// ---- ECC/Basic/TrackClient/Node Data/ST_ReadStationData.TcDUT
{attribute 'pack_mode' := '1'}
TYPE ST_ReadStationData :
STRUCT
	stReadListReturnInfo		: ARRAY [1..1] OF ST_UAReadListReturnInfo;
	stStationData				: ST_StatusStation;

END_STRUCT
END_TYPE

// ---- ECC/Basic/TrackClient/Node Data/ST_ReadVehicleData.TcDUT
{attribute 'pack_mode' := '1'}
TYPE ST_ReadVehicleData :
STRUCT
	stReadListReturnInfo		: ARRAY [1..1] OF ST_UAReadListReturnInfo;
	stVehicle					: ST_StatusVehicle;

END_STRUCT
END_TYPE

// ---- ECC/Basic/TrackClient/Node Data/ST_ReadVehicleData_OLD.TcDUT
{attribute 'pack_mode' := '1'}
TYPE ST_ReadVehicleData_OLD :
STRUCT
//	stReadListReturnInfo		: ARRAY [1..1] OF ST_UAReadListReturnInfo;
//	stVehicle					: ST_StatusVehicle;

	// Array must have the same number as the amount of elements in the status strucuture! 
	stReadListReturnInfo		: ARRAY [1..8] OF ST_UAReadListReturnInfo;
	nVehicleID					: UINT;
	bVehiclePresent				: BOOL;
	nState						: UINT; 
	nPathID						: UINT;
	fPosition					: REAL;
	nTargetPathID				: UINT;
	fTargetPosition				: REAL;
	fVelocity					: REAL;
END_STRUCT
END_TYPE

// ---- ECC/Basic/TrackClient/Node Data/ST_StatusCell.TcDUT
/// Standard Status for cells
TYPE ST_StatusCell :
STRUCT
	sCellID						: STRING(30);		(*  *)
	sNextCellOnTrack			: STRING(30);		(*  *)
//	nVehicleIDDecisionPoint		: UINT;				(* ID of the vehicle ready at cell decision point *)
//													(* ZERO of no vehicle is ready *)	
//	sCarrierIDDecisionPoint		: STRING(30);		(* ID of the carrier ready at cell decision point *)
	astReservations				: ARRAY [1..MM_MAX_RESERVATIONLIST_ELEMENTS] OF ST_ReservationData; (* Reservation lists for cells. *)
																									(* NOTE! Only manipulated through methods M_AddReservationList, M_RemoveReservationList *)
	anVehicles					: ARRAY [1..MM_MAX_NUMBER_OF_VEHICLE_ELEMENTS] OF UINT;				(* Vehicles ID's of the vehicles controlled by this cell *)

END_STRUCT
END_TYPE

// ---- ECC/Basic/TrackClient/Node Data/ST_StatusNode.TcDUT
{attribute 'pack_mode' := '1'}
TYPE ST_StatusNode :
STRUCT
	nState	: UINT;
	rTemp	: REAL;
END_STRUCT
END_TYPE

// ---- ECC/Basic/TrackClient/Node Data/ST_StatusPath.TcDUT
{attribute 'pack_mode' := '1'}
TYPE ST_StatusPath :
STRUCT
	nPathID						: UINT;
	sCellID						: STRING(30);
	bPathPresent				: BOOL;
	nState						: UINT;			// E_MMPathState
	nMotionStatus				: UINT;			// E_MMPathMotionStatus
END_STRUCT
END_TYPE

// ---- ECC/Basic/TrackClient/Node Data/ST_StatusStation.TcDUT
{attribute 'pack_mode' := '1'}
TYPE ST_StatusStation :
STRUCT
	sCellID						: STRING(30);
	sStationID					: STRING(30);
	bStationPresent				: BOOL;
	nVehicleIDDecisionPoint		: UINT;				(* ID of the vehicle ready at station decision point. ZERO of no vehicle is ready *)	
	sCarrierIDDecisionPoint		: STRING(30);		(* ID of the carrier ready at station decision point *)
	nVehicleIDStationIn			: UINT;				(* ID of the vehicle ready at station location In location. ZERO of no vehicle is ready *)	
	sCarrierIDStationIn			: STRING(30);		(* ID of the carrier ready at station location In location *)
	nVehicleIDStationOut		: UINT;				(* ID of the vehicle ready at station location Out ZERO of no vehicle is ready *)	
	sCarrierIDStationOut		: STRING(30);		(* ID of the carrier ready at station location Out location *)
//	stStation					: ST_StatusBuffer;
//	aPreBuffer					: ARRAY [1..MM_MAX_BUFFER_INDEX] OF ST_StatusBuffer;
//	aPostBuffer					: ARRAY [1..MM_MAX_BUFFER_INDEX] OF ST_StatusBuffer;

END_STRUCT
END_TYPE

// ---- ECC/Basic/TrackClient/Node Data/ST_StatusVehicle.TcDUT
{attribute 'pack_mode' := '1'}
TYPE ST_StatusVehicle :
STRUCT
	nVehicleID					: UINT;
	sOwnerCell					: STRING(30);				// Cell which controls this vehicle
	nState						: UINT;						// E_CarrierStatus: 0: Undefined, 1: Initiating, 2: Not Busy(No Ticket), 3: Busy(Ticket), 4: Montage Reserved
	bVehiclePresent				: BOOL;
	bDataValid					: BOOL;
	sLastScan					: STRING(30);				// Timestamp for last scan of this vehicle
	sCarrierID					: STRING(30);				// Scanned (from Carrier RFID scan)
	bTool						: BOOL;						// TRUE if tool is mounted on carrier
	sToolID						: STRING(30);				// Tool ID (if mounted) (from Tool RFID scan)
	bMaterial					: BOOL;						// TRUE if material is mounted on Tray (tool)
	sMaterialID					: STRING(30);				// Optional, Mterial ID (from material RFID scan)
	sJobID						: STRING(30);				// Job ID assigned to this vehicle/carrier
	nTicket						: UINT;						// Ticket for item on this vehicle
	nTicketSize					: UINT;						// Size of ticket (carriers in package)
	nPriority					: UINT;						// Priority within ticket
	nPathID						: UINT;						// Current path
	fPosition					: REAL;						// Current location on the path
	nTargetPathID				: UINT;						// Target path
	fTargetPosition				: REAL;						// Target location on target path
	fVelocity					: REAL;						// Actual velocity
	sTargetStationID			: STRING(30);				// Target station
	sCurrentStationID			: STRING(30);				// Actual station
	bNOK						: BOOL;						// TRUE of rework is required

END_STRUCT
END_TYPE

// ---- ECC/Basic/TrackClient/Node Data/SUB/ST_ReservationData.TcDUT
TYPE ST_ReservationData :
STRUCT
	bUsed					: BOOL;
	nTicket					: UINT;														(*  *)
	nTicketSize				: UINT;														(*  *)
	sStationID				: STRING(30);												(*  *)
	sAddedTime				: STRING(30);												(* Date and time for when entry was added *)
END_STRUCT
END_TYPE

// ---- ECC/Basic/TrackClient/OPC Data/ST_InputTransport.TcDUT
TYPE ST_InputTransport :
STRUCT
	{attribute 'OPC.UA.DA.Description' := 'Track command data'}
	{attribute 'OPC.UA.DA.StructuredType' := '1'}
	{attribute 'TcIgnorePersistent'}
	Command				: ST_InputTransportCommand;
	
	{attribute 'OPC.UA.DA.Description' := 'Track mapping data'}
	{attribute 'OPC.UA.DA.StructuredType' := '1'}
	Mapping				: ST_InputTransportMapping;
	
	{attribute 'OPC.UA.DA.Description' := 'Track configuration data'}
	{attribute 'OPC.UA.DA.StructuredType' := '1'}
	Configuration		: ST_InputTransportConfiguration;
	
	{attribute 'OPC.UA.DA.Description' := 'Track additional data'}
	{attribute 'OPC.UA.DA.StructuredType' := '1'}
	{attribute 'TcIgnorePersistent'}
	AdditionalData		: ST_InputTransportAdditionalData;
	
END_STRUCT
END_TYPE

// ---- ECC/Basic/TrackClient/OPC Data/ST_OutputTransport.TcDUT
TYPE ST_OutputTransport :
STRUCT
	{attribute 'OPC.UA.DA.Description' := 'Track status data'}
	{attribute 'OPC.UA.DA.StructuredType' := '1'}
	Status				: ST_OutputTransportStatus;
	
	{attribute 'OPC.UA.DA.Description' := 'Track mapping data'}
	{attribute 'OPC.UA.DA.StructuredType' := '1'}
	Mapping				: ST_OutputTransportMapping;
	
	{attribute 'OPC.UA.DA.Description' := 'Track configuration data'}
	{attribute 'OPC.UA.DA.StructuredType' := '1'}
	Configuration		: ST_OutputTransportConfiguration;
	
	{attribute 'OPC.UA.DA.Description' := 'Track additional data'}
	{attribute 'OPC.UA.DA.StructuredType' := '1'}
	AdditionalData		: ST_OutputTransportAdditionalData;
	
END_STRUCT
END_TYPE

// ---- ECC/Basic/TrackClient/OPC Data/Sub/ST_BufferIndexX.TcDUT
TYPE ST_BufferIndexX :
STRUCT
	{attribute 'OPC.UA.DA.Description' := 'TRUE if carrier is on the index'}
	Present					: BOOL;

	{attribute 'OPC.UA.DA.Description' := 'Ticket for the carrier on the index (0-65536)'}
	Ticket					: UINT;

	{attribute 'OPC.UA.DA.Description' := 'Carrier ID fir the carrier in the index'}
	CarrierID				: STRING(30);

END_STRUCT
END_TYPE

// ---- ECC/Basic/TrackClient/OPC Data/Sub/ST_CarrierX.TcDUT
TYPE ST_CarrierX :
STRUCT
	{attribute 'OPC.UA.DA.Description' := 'Carrier ID'}
	CarrierID					: STRING(30);
	
	{attribute 'OPC.UA.DA.Description' := 'Carrier status (0: Undefined, 1: Initiating, 2: Not busy, 3: Busy)'}
	CarrierStatus				: UINT;

	{attribute 'OPC.UA.DA.Description' := 'Status data are valid'}
	ValidData					: BOOL;

	{attribute 'OPC.UA.DA.Description' := 'Date and time of the last scan of this carrier'}
	LastScan					: DT;

	{attribute 'OPC.UA.DA.Description' := 'TRUE if a tool is mounted on the carrier'}
	Tool						: BOOL;

	{attribute 'OPC.UA.DA.Description' := 'Tool ID'}
	ToolID						: STRING(30);

	{attribute 'OPC.UA.DA.Description' := 'TRUE if material is mounted on the carrier'}
	Material					: BOOL;

	{attribute 'OPC.UA.DA.Description' := 'Material ID'}
	MaterialID					: STRING(30);

	{attribute 'OPC.UA.DA.Description' := 'SKU ID'}
	JobID						: STRING(30);

	{attribute 'OPC.UA.DA.Description' := 'Packet (Ticket) (0-65536)'}
	Ticket						: UINT;
	
	{attribute 'OPC.UA.DA.Description' := 'Carriers in packet (Ticket) (0-100)'}
	CarriersInPackage			: UINT;

	{attribute 'OPC.UA.DA.Description' := 'Priority within the packet (ticket)'}
	Priority					: UINT;
	
	{attribute 'OPC.UA.DA.Description' := 'Current location, Path ID'}
	CurrentPath					: UINT;

	{attribute 'OPC.UA.DA.Description' := 'Current location, Position on path (mm)'}
	CurrentPosition				: REAL;

	{attribute 'OPC.UA.DA.Description' := 'Current station for this carrier'}
	CurrentStation				: STRING(30);

	{attribute 'OPC.UA.DA.Description' := 'Target station for this carrier'}
	TargetStation				: STRING(30);

	{attribute 'OPC.UA.DA.Description' := 'Target reached for this carrier'}
	TargetReached				: BOOL;

	{attribute 'OPC.UA.DA.Description' := 'Target reached counter for this carrier'}
	TargetReachedCounter		: UINT;

	{attribute 'OPC.UA.DA.Description' := 'Indicator for Not OK'}
	NOK							: BOOL;

END_STRUCT
END_TYPE

// ---- ECC/Basic/TrackClient/OPC Data/Sub/ST_InputTransportAdditionalData.TcDUT
TYPE ST_InputTransportAdditionalData :
STRUCT
	{attribute 'OPC.UA.DA.Description' := 'Transport MES handshakes'}
	{attribute 'OPC.UA.DA.StructuredType' := '1'}
	MESHandShakes				: ST_InputTransportAdditionalDataMESHandShake;

	{attribute 'OPC.UA.DA.Description' := 'Transport MES Handshakes'}
	{attribute 'OPC.UA.DA.StructuredType' := '1'}
	Settings					: ST_InputTransportAdditionalDataSettings;
	
	{attribute 'OPC.UA.DA.Description' := 'Exit point ticket release delay (s)'}
	ExitPointReleaseDelay		: REAL := 0.0;
	
	{attribute 'OPC.UA.DA.Description' := 'Allow initilization on Track Server (Create Stations etc.)'}
	bAllowInit					: BOOL;		// TRUE to allow initilization to track server (create Stations, DecisionPoint, TrafficLight etc. to Track Server)

	{attribute 'OPC.UA.DA.Description' := 'Set to TRUE to shut down the track on this cell'}
	bShutDown					: BOOL;

END_STRUCT
END_TYPE

// ---- ECC/Basic/TrackClient/OPC Data/Sub/ST_InputTransportAdditionalDataMESHandShake.TcDUT
TYPE ST_InputTransportAdditionalDataMESHandShake :
STRUCT
	{attribute 'OPC.UA.DA.Description' := 'Data Change status for Status values (0-65536)'}
	DataChangeStatusTransportStatus		: UINT;

	{attribute 'OPC.UA.DA.Description' := 'Data Change status for Mapping values (0-65536)'}
	DataChangeStatusTransportMapping	: UINT;

END_STRUCT
END_TYPE

// ---- ECC/Basic/TrackClient/OPC Data/Sub/ST_InputTransportAdditionalDataSettings.TcDUT
TYPE ST_InputTransportAdditionalDataSettings :
STRUCT
	{attribute 'OPC.UA.DA.Description' := 'Transport Status update Enable'}
	DataChangeStatusTransportStatusEnable	: BOOL;

	{attribute 'OPC.UA.DA.Description' := 'Transport Mapping update Enable'}
	DataChangeStatusTransportMappingEnable	: BOOL;

END_STRUCT
END_TYPE

// ---- ECC/Basic/TrackClient/OPC Data/Sub/ST_InputTransportCommand.TcDUT
TYPE ST_InputTransportCommand :
STRUCT
	{attribute 'OPC.UA.DA.Description' := 'Change Request (0-255)'}
	ChangeRequest			: UINT;

	{attribute 'OPC.UA.DA.Description' := 'Carrier ID'}
	CarrierID				: STRING(30);

	{attribute 'OPC.UA.DA.Description' := 'Packet (Ticket) ID (1-65536)'}
	Ticket					: UINT;

	{attribute 'OPC.UA.DA.Description' := 'Number of carriers in Packet (Ticket) (1-100)'}
	CarriersInPackage		: UINT;

	{attribute 'OPC.UA.DA.Description' := 'Priority within Packet (Ticket) (1-100)'}
	Priority				: UINT;

	{attribute 'OPC.UA.DA.Description' := 'Assigned Job ID'}
	JobID					: STRING(30);

	{attribute 'OPC.UA.DA.Description' := 'Target station ID'}
	TargetStation			: STRING(30);
	
END_STRUCT
END_TYPE

// ---- ECC/Basic/TrackClient/OPC Data/Sub/ST_InputTransportConfiguration.TcDUT
TYPE ST_InputTransportConfiguration :
STRUCT
	{attribute 'OPC.UA.DA.Description' := 'Location for decision point'}
	{attribute 'OPC.UA.DA.StructuredType' := '1'}
	DecisionPointLocation		: ST_TrackLocation;

	{attribute 'OPC.UA.DA.Description' := 'Location for traffic light'}
	{attribute 'OPC.UA.DA.StructuredType' := '1'}
	TrafficLightLocation		: ST_TrackLocation;
	
	{attribute 'OPC.UA.DA.Description' := 'Location for traffic light'}
	{attribute 'OPC.UA.DA.StructuredType' := '1'}
	Stations					: ARRAY [1..5] OF ST_StationConfigX;

END_STRUCT
END_TYPE

// ---- ECC/Basic/TrackClient/OPC Data/Sub/ST_InputTransportMapping.TcDUT
TYPE ST_InputTransportMapping :
STRUCT
	{attribute 'OPC.UA.DA.Description' := 'Change Request (0-255)'}
	ChangeRequest			: UINT;
	
	{attribute 'OPC.UA.DA.Description' := 'Track carrier mapping data'}
	{attribute 'OPC.UA.DA.StructuredType' := '1'}
	Carrier					: ST_TransportMappingCarrier;
	
	{attribute 'OPC.UA.DA.Description' := 'Track station mapping data'}
	{attribute 'OPC.UA.DA.StructuredType' := '1'}
	StationBuffer			: ST_TransportMappingStationBuffer;

END_STRUCT
END_TYPE

// ---- ECC/Basic/TrackClient/OPC Data/Sub/ST_OutputTransportAdditionalData.TcDUT
TYPE ST_OutputTransportAdditionalData :
STRUCT
	{attribute 'OPC.UA.DA.Description' := 'TRUE if Track Client is connected to Track Server for method calls'}
	bConnectedMethod			: BOOL;

	{attribute 'OPC.UA.DA.Description' := 'TRUE if Track Client is connected to Track Server for data reading'}
	bConnectedNode				: BOOL;

	{attribute 'OPC.UA.DA.Description' := 'TRUE if Track Client is ready to work (DecisionPoint, ExitPoint, Buffers)'}
	bTrackReady					: BOOL;

END_STRUCT
END_TYPE

// ---- ECC/Basic/TrackClient/OPC Data/Sub/ST_OutputTransportConfiguration.TcDUT
TYPE ST_OutputTransportConfiguration :
STRUCT
	{attribute 'OPC.UA.DA.Description' := 'Dummy (for making struct visible on OPC UA'}
	Dummy						: BOOL;

END_STRUCT
END_TYPE

// ---- ECC/Basic/TrackClient/OPC Data/Sub/ST_OutputTransportMapping.TcDUT
TYPE ST_OutputTransportMapping :
STRUCT
// Handshake part
	{attribute 'OPC.UA.DA.Description' := 'Change acknowledge (0-255)'}
	ChangeAcknowlegde		: UINT;						// Indicator to acknowledge that a new mapping will be handled
	
	{attribute 'OPC.UA.DA.Description' := 'Change status (0-255)'}
	ChangeStatus			: UINT;						// Indicator that a new mapping has been handled
	
// Data part
	{attribute 'OPC.UA.DA.Description' := 'Data Change (0-65535)'}
	DataChange				: UINT;						// Indicator that output variables in Mapping has been updated
	
	{attribute 'OPC.UA.DA.Description' := 'The request is valid'}
	ValidRequest				: BOOL;

	{attribute 'OPC.UA.DA.Description' := 'Track carrier mapping data'}
	{attribute 'OPC.UA.DA.StructuredType' := '1'}
	Carrier					: ST_TransportMappingCarrier;	// 
	
	{attribute 'OPC.UA.DA.Description' := 'Track station mapping data'}
	{attribute 'OPC.UA.DA.StructuredType' := '1'}
	StationBuffer			: ST_TransportMappingStationBuffer;	// 

END_STRUCT
END_TYPE

// ---- ECC/Basic/TrackClient/OPC Data/Sub/ST_OutputTransportStatus.TcDUT
TYPE ST_OutputTransportStatus :
STRUCT
// Handshake part
	{attribute 'OPC.UA.DA.Description' := 'Change Acknowledge (0-255)'}
	ChangeAcknowledge			: UINT;

	{attribute 'OPC.UA.DA.Description' := 'Change Status (0-255)'}
	ChangeStatus				: UINT;

// Data part
	{attribute 'OPC.UA.DA.Description' := 'Data Changed (0-65536)'}
	DataChange					: UINT;

	{attribute 'OPC.UA.DA.Description' := 'The request is valid'}
	ValidRequest				: BOOL;

	{attribute 'OPC.UA.DA.Description' := 'Last handled ticket (0-65536)'}
	LatestTicket				: UINT;

	{attribute 'OPC.UA.DA.Description' := 'Number of carriers under this bridge responsibility (0-1000)'}
	NumberOfCarriers			: UINT;

	{attribute 'OPC.UA.DA.Description' := 'Carrier Status'}
	{attribute 'OPC.UA.DA.StructuredType' := '1'}
	Carrier						: ARRAY [1..1000] OF ST_CarrierX;

	{attribute 'OPC.UA.DA.Description' := 'Station buffer Status'}
	{attribute 'OPC.UA.DA.StructuredType' := '1'}
	StationBuffer				: ARRAY [1..5] OF ST_StationBufferX;

END_STRUCT
END_TYPE

// ---- ECC/Basic/TrackClient/OPC Data/Sub/ST_StationBufferStatus.TcDUT
TYPE ST_StationBufferStatus :
STRUCT
	{attribute 'OPC.UA.DA.Description' := 'Capacity (0-100)'}
	Capacity				: UINT;
	
	{attribute 'OPC.UA.DA.Description' := 'Capacity used (0-100)'}
	CapacityUsed			: UINT;

	{attribute 'OPC.UA.DA.Description' := 'Buffer status data'}
	{attribute 'OPC.UA.DA.StructuredType' := '1'}
	BufferIndex				: ARRAY [1..100] OF ST_BufferIndexX;

END_STRUCT
END_TYPE

// ---- ECC/Basic/TrackClient/OPC Data/Sub/ST_StationBufferX.TcDUT
TYPE ST_StationBufferX :
STRUCT
	{attribute 'OPC.UA.DA.Description' := 'Station ID'}
	StationID					: STRING(30);

	{attribute 'OPC.UA.DA.Description' := 'Pre buffer'}
	{attribute 'OPC.UA.DA.StructuredType' := '1'}
	PreBuffer					: ST_StationBufferStatus;
	
	{attribute 'OPC.UA.DA.Description' := 'Post buffer'}
	{attribute 'OPC.UA.DA.StructuredType' := '1'}
	PostBuffer					: ST_StationBufferStatus;

END_STRUCT
END_TYPE

// ---- ECC/Basic/TrackClient/OPC Data/Sub/ST_StationConfigX.TcDUT
TYPE ST_StationConfigX :
STRUCT
	{attribute 'OPC.UA.DA.Description' := 'Station ID'}
	StationID					: STRING(30);

	{attribute 'OPC.UA.DA.Description' := 'Station location'}
	{attribute 'OPC.UA.DA.StructuredType' := '1'}
	StationLocation1			: ST_TrackLocation;

	{attribute 'OPC.UA.DA.Description' := 'Station location'}
	{attribute 'OPC.UA.DA.StructuredType' := '1'}
	StationLocation2			: ST_TrackLocation;

	{attribute 'OPC.UA.DA.Description' := 'Decision Point location'}
	{attribute 'OPC.UA.DA.StructuredType' := '1'}
	DecisionPointLocation		: ST_TrackLocation;

	{attribute 'OPC.UA.DA.Description' := 'Pre buffer size (0-10)'}
	PreBufferSize				: UINT;
	
	{attribute 'OPC.UA.DA.Description' := 'Post buffer size (0-10)'}
	PostBufferSize				: UINT;

END_STRUCT
END_TYPE

// ---- ECC/Basic/TrackClient/OPC Data/Sub/ST_StatusBuffer.TcDUT
TYPE ST_StatusBuffer :
STRUCT
	bPresent		: BOOL;		// TRUE if buffer point is in use
	nTicket			: UINT;		// Reseved Ticket ID 
	nPriority		: UINT;		// Current Ticket priority
	nVehicleID		: UINT;		// Current vehicle ID (0 if no vehicle)
END_STRUCT
END_TYPE

// ---- ECC/Basic/TrackClient/OPC Data/Sub/ST_TrackLocation.TcDUT
TYPE ST_TrackLocation :
STRUCT
	{attribute 'OPC.UA.DA.Description' := 'Location path (ID)'}
	Path			: UINT;

	{attribute 'OPC.UA.DA.Description' := 'Location position (m)'}
	Position		: REAL;
	
END_STRUCT
END_TYPE

// ---- ECC/Basic/TrackClient/OPC Data/Sub/ST_TransportMappingCarrier.TcDUT
TYPE ST_TransportMappingCarrier :
STRUCT
	{attribute 'OPC.UA.DA.Description' := 'Carrier ID'}
	CarrierID					: STRING(30);			// Unique ID of the Carrier which the change is aimed towards. If CarrierID is 0 there is no Mapping information to update

	{attribute 'OPC.UA.DA.Description' := 'Tool ?'}
	Tool						: BOOL;					// Indicates if there is a Tool or not on the carrirer, 0 = No tool, 1 = Tool
	
	{attribute 'OPC.UA.DA.Description' := 'Tool ID'}
	ToolID						: STRING(30);			// Mandatory if Tool = 1. Unique ID(UUID) of the tool to be mapped with defined CarrierID
	
	{attribute 'OPC.UA.DA.Description' := 'Material ?'}
	Material					: BOOL;					// Indicates if there is a Material or not related to the carrirer, 0 = No material, 1 = Material
	
	{attribute 'OPC.UA.DA.Description' := 'Material ID'}
	MaterialID					: STRING(30);			// Mandatory if Material = 1. Unique ID(UUID) of the Material to be mapped with defined CarrierID
	
	{attribute 'OPC.UA.DA.Description' := 'Not OK'}
	NOK							: BOOL;					// “0” = No change to Carrier Status. “1” = Carrier must be flagged with “NOK” and the “NOK” procedure gets triggered.
	
	{attribute 'OPC.UA.DA.Description' := 'Data is valid'}
	ValidData					: BOOL;					// Indicator that the variables for carrier can be considered valid.
	
END_STRUCT
END_TYPE

// ---- ECC/Basic/TrackClient/OPC Data/Sub/ST_TransportMappingStationBuffer.TcDUT
TYPE ST_TransportMappingStationBuffer :
STRUCT
	{attribute 'OPC.UA.DA.Description' := 'Dummy (for making struct visible on OPC UA'}
	Dummy						: BOOL;

END_STRUCT
END_TYPE

// ---- ECC/Cell_Unit_4/E_VehicleOnStation.TcDUT
{attribute 'qualified_only'}
{attribute 'strict'}
TYPE E_VehicleOnStation :
(
	Idle := 0,
	VehicleAtStation,
	AddToFIFO,
	WaitStationStart,
	MoveVehicle,
	VehicleLeftStation
);
END_TYPE

// ---- ECC/Cell_Unit_4/HeatAndSteamDeviceDriver/Sub/E_EMS_HS_Status.TcDUT
{attribute 'qualified_only'}
{attribute 'strict'}
TYPE E_EMS_HS_Status :
(
	STANDBY := 0,	// Stand-by - Not ready to work
	PREPARING,		// Preparing - Not ready to work
	READY,			// Ready to work
	ALARM			// Alarm!

);
END_TYPE

// ---- ECC/Cell_Unit_4/HeatAndSteamDeviceDriver/Sub/ST_EMS_HS_Alarms.TcDUT
{attribute 'pack_mode' := '1'}
TYPE ST_EMS_HS_Alarms :
STRUCT
	TEMP_PROBE_FAULT		: BIT;	// BIT 0
	FAULT_INVERTER			: BIT;	// BIT 1
	{attribute 'OPC.UA.DA':='0'}
	DISP_2					: BIT;	// BIT 2
	{attribute 'OPC.UA.DA':='0'}
	DISP_3					: BIT;	// BIT 3
	{attribute 'OPC.UA.DA':='0'}
	DISP_4					: BIT;	// BIT 4
	{attribute 'OPC.UA.DA':='0'}
	DISP_5					: BIT;	// BIT 5
	ENERGY_METER_COM_ERROR	: BIT;	// BIT 6
	{attribute 'OPC.UA.DA':='0'}
	DISP_7					: BIT;	// BIT 7
	{attribute 'OPC.UA.DA':='0'}
	DISP_8					: BIT;	// BIT 8
	{attribute 'OPC.UA.DA':='0'}
	DISP_9					: BIT;	// BIT 9
	{attribute 'OPC.UA.DA':='0'}
	DISP_10					: BIT;	// BIT 10
	{attribute 'OPC.UA.DA':='0'}
	DISP_11					: BIT;	// BIT 11
	{attribute 'OPC.UA.DA':='0'}
	DISP_12					: BIT;	// BIT 12
	{attribute 'OPC.UA.DA':='0'}
	DISP_13					: BIT;	// BIT 13
	{attribute 'OPC.UA.DA':='0'}
	DISP_14					: BIT;	// BIT 14
	{attribute 'OPC.UA.DA':='0'}
	DISP_15					: BIT;	// BIT 15

END_STRUCT
END_TYPE

// ---- ECC/Cell_Unit_4/HeatAndSteamDeviceDriver/Sub/ST_EMS_HS_Command.TcDUT
{attribute 'pack_mode' := '1'}
TYPE ST_EMS_HS_Command :
STRUCT
	REMOTE_START			: BIT;	// BIT 0
	REMOTE_STOP				: BIT;	// BIT 1
	{attribute 'OPC.UA.DA':='0'}
	DISP_2					: BIT;	// BIT 2
	RESET_RUNNING_HRS		: BIT;	// BIT 3
	RESET_ENERGY_CONS		: BIT;	// BIT 4
	{attribute 'OPC.UA.DA':='0'}
	DISP_5					: BIT;	// BIT 5
	{attribute 'OPC.UA.DA':='0'}
	DISP_6					: BIT;	// BIT 6
	{attribute 'OPC.UA.DA':='0'}
	DISP_7					: BIT;	// BIT 7	
	{attribute 'OPC.UA.DA':='0'}
	DISP_8					: BIT;	// BIT 8
	{attribute 'OPC.UA.DA':='0'}
	DISP_9					: BIT;	// BIT 9
	{attribute 'OPC.UA.DA':='0'}
	DISP_10					: BIT;	// BIT 10
	{attribute 'OPC.UA.DA':='0'}
	DISP_11					: BIT;	// BIT 11
	{attribute 'OPC.UA.DA':='0'}
	DISP_12					: BIT;	// BIT 12
	{attribute 'OPC.UA.DA':='0'}
	DISP_13					: BIT;	// BIT 13	
	{attribute 'OPC.UA.DA':='0'}
	DISP_14					: BIT;	// BIT 14	
	{attribute 'OPC.UA.DA':='0'}
	DISP_15					: BIT;	// BIT 15	

END_STRUCT
END_TYPE

// ---- ECC/Cell_Unit_4/HeatAndSteamDeviceDriver/Sub/ST_EMS_HS_Read.TcDUT
 {attribute 'pack_mode' := '1'}
TYPE ST_EMS_HS_Read :
STRUCT
	{attribute 'OPC.UA.DA.Description' := 'Actual temperature value'}
	rActTempVal			: REAL;								// [°C] - 32bit float - addr:2501
	{attribute 'OPC.UA.DA.Description' := 'Actual desired temperature'}
	rActTempSetpoint	: REAL;								// [°C] - 32bit float - addr:2503
	{attribute 'OPC.UA.DA.Description' := 'Actual steam request'}
	rActSteamReq		: DINT;								// [] - 32bit float - addr:2505
	{attribute 'OPC.UA.DA.Description' := 'Actual fan speed request'}
	rActFanReq			: REAL;								// [RPM] - 32bit float - addr:2507
	{attribute 'OPC.UA.DA.Description' := 'Instant power'}
	rInstPower			: REAL;								// [kW] - 32bit float - addr:2509
	{attribute 'OPC.UA.DA.Description' := 'Energy consumption'}
	rEnergyCons			: REAL;								// [kWh] - 32bit float - addr:2511
	{attribute 'OPC.UA.DA.Description' := 'Running hours'}
	iRunningHrs			: UDINT;							// [hours] - 32bit udint - addr:2513
	{attribute 'OPC.UA.DA.Description' := 'Running minutes'}
	iRunningMins		: UDINT;							// [minutes] - 32bit udint - addr:2515
	{attribute 'OPC.UA.DA':='0'}
	{attribute 'hide'}
	wDisp2017			: WORD;
	{attribute 'OPC.UA.DA':='0'}
	{attribute 'hide'}
	wDisp2018			: WORD;
	{attribute 'OPC.UA.DA':='0'}
	{attribute 'hide'}
	wDisp2019			: WORD;
	{attribute 'OPC.UA.DA':='0'}
	{attribute 'hide'}
	wDisp2020			: WORD;
	{attribute 'OPC.UA.DA.Description' := 'Station status'}
	eMachStatus			: E_EMS_HS_Status;	// - 16bit uint - addr:2521
	{attribute 'OPC.UA.DA.Description' := 'Station status bits'}
	stStates			: ST_EMS_HS_States;	// - 16bit word - addr:2522
	{attribute 'OPC.UA.DA.Description' := 'Station alarms bits'}
	stAlarms			: ST_EMS_HS_Alarms;	// - 16bit word	 - addr:2523
	
END_STRUCT
END_TYPE

// ---- ECC/Cell_Unit_4/HeatAndSteamDeviceDriver/Sub/ST_EMS_HS_States.TcDUT
{attribute 'pack_mode' := '1'}
TYPE ST_EMS_HS_States :
STRUCT
	REMOTE_MODE				: BIT;	// BIT 0
	ALARM_IN_PROGRESS		: BIT;	// BIT 1
	MACHINE_READY_TO_WORK	: BIT;	// BIT 2
	TEMP_START_BELT_REACHED	: BIT;	// BIT 3
	TEMP_START_STEAM_REACHED: BIT;	// BIT 4
	MACHINE_IN_STANDBY		: BIT;	// BIT 5
	MACHINE_IN_HEATING		: BIT;	// BIT 6
	{attribute 'OPC.UA.DA':='0'}
	DISP_7					: BIT;	// BIT 7
	{attribute 'OPC.UA.DA':='0'}
	DISP_8					: BIT;	// BIT 8
	{attribute 'OPC.UA.DA':='0'}
	DISP_9					: BIT;	// BIT 9
	{attribute 'OPC.UA.DA':='0'}
	DISP_10					: BIT;	// BIT 10
	{attribute 'OPC.UA.DA':='0'}
	DISP_11					: BIT;	// BIT 11
	{attribute 'OPC.UA.DA':='0'}
	DISP_12					: BIT;	// BIT 12
	{attribute 'OPC.UA.DA':='0'}
	DISP_13					: BIT;	// BIT 13
	{attribute 'OPC.UA.DA':='0'}
	DISP_14					: BIT;	// BIT 14
	{attribute 'OPC.UA.DA':='0'}
	DISP_15					: BIT;	// BIT 15

END_STRUCT
END_TYPE

// ---- ECC/Cell_Unit_4/HeatAndSteamDeviceDriver/Sub/ST_EMS_HS_Write.TcDUT
{attribute 'pack_mode' := '1'}
TYPE ST_EMS_HS_Write :
STRUCT
	{attribute 'OPC.UA.DA.Description' := 'Station commands'}
	stCommands			: ST_EMS_HS_Command;	// - 16bit word - addr:2601
	{attribute 'OPC.UA.DA':='0'}
	{attribute 'hide'}
	Disp2602			: WORD;
	{attribute 'OPC.UA.DA.Description' := 'Remote desired temperature'}
	rSetTemp			: REAL;								// [°C] - 32bit float - addr:2603
	{attribute 'OPC.UA.DA.Description' := 'Remote desired steam request'}
	rSetSteamReq		: DINT;								// [0-10] - 32bit float - addr:2605
	{attribute 'OPC.UA.DA.Description' := 'Remote desired fan speed'}
	rSetFanSpeed		: REAL;								// [RPM] - 32bit float - addr:2607
	
END_STRUCT
END_TYPE

// ---- ECC/Cell_Unit_4/HeatAndSteamDeviceDriver/U_EMS_HS_Read.TcDUT
TYPE U_EMS_HS_Read :
UNION
	aWords					: ARRAY [1..23] OF WORD;
	stVars					: ST_EMS_HS_Read;

END_UNION
END_TYPE

// ---- ECC/Cell_Unit_4/HeatAndSteamDeviceDriver/U_EMS_HS_Write.TcDUT
TYPE U_EMS_HS_Write :
UNION
	aWords					: ARRAY [1..8] OF WORD;
	stVars					: ST_EMS_HS_Write;

END_UNION
END_TYPE

// ---- ECC/Cell_Unit_4/HeatAndSteam/OPC Data/Sub/AdditionalData/ST_InputStationHSAdditionalDataOP11600.TcDUT
TYPE ST_InputStationHSAdditionalDataOP11600 :
STRUCT
	{attribute 'OPC.UA.DA.Description' := 'Initial Temperature'}
	TempInitial					: REAL := 20.0;

END_STRUCT
END_TYPE

// ---- ECC/Cell_Unit_4/HeatAndSteam/OPC Data/Sub/AdditionalData/ST_InputStationHSAdditionalDataOP11601.TcDUT
TYPE ST_InputStationHSAdditionalDataOP11601 :
STRUCT
	{attribute 'OPC.UA.DA.Description' := 'Dummy (for making struct visible on OPC UA'}
	Dummy						: BOOL;
END_STRUCT
END_TYPE

// ---- ECC/Cell_Unit_4/HeatAndSteam/OPC Data/Sub/AdditionalData/ST_InputStationHSAdditionalDataMESHandShake.TcDUT
TYPE ST_InputStationHSAdditionalDataMESHandShake :
STRUCT
	{attribute 'OPC.UA.DA.Description' := 'Station ModeState update status'}
	{attribute 'TcIgnorePersistent'}
	DataChangeStatusModeState				: UINT;

	{attribute 'OPC.UA.DA.Description' := 'Station Job Data update status'}
	{attribute 'TcIgnorePersistent'}
	DataChangeStatusJobData					: UINT;

	{attribute 'OPC.UA.DA.Description' := 'Station OEE update status'}
	{attribute 'TcIgnorePersistent'}
	DataChangeStatusOEE						: UINT;

	{attribute 'OPC.UA.DA.Description' := 'Station ErrorWarning update status'}
	{attribute 'TcIgnorePersistent'}
	DataChangeStatusErrorWarning			: UINT;

	{attribute 'OPC.UA.DA.Description' := 'Station Current Configuration update status'}
	{attribute 'TcIgnorePersistent'}
	DataChangeStatusCurrentConfiguration	: UINT;

	{attribute 'OPC.UA.DA.Description' := 'Station Upcoming Configuration update status'}
	{attribute 'TcIgnorePersistent'}
	DataChangeStatusUpcomingConfiguration	: UINT;

	{attribute 'OPC.UA.DA.Description' := 'Station Operationaldata update status'}
	{attribute 'TcIgnorePersistent'}
	DataChangeStatusOperationalData			: UINT;

END_STRUCT
END_TYPE

// ---- ECC/Cell_Unit_4/HeatAndSteam/OPC Data/Sub/AdditionalData/ST_InputStationHSAdditionalDataSettings.TcDUT
TYPE ST_InputStationHSAdditionalDataSettings :
STRUCT
	{attribute 'OPC.UA.DA.Description' := 'Station ModeState update Enable'}
	DataChangeStatusModeStateEnable				: BOOL;

	{attribute 'OPC.UA.DA.Description' := 'Station JobData update Enable'}
	DataChangeStatusJobDataEnable				: BOOL;

	{attribute 'OPC.UA.DA.Description' := 'Station OEE update Enable'}
	DataChangeStatusOEEEnable					: BOOL;

	{attribute 'OPC.UA.DA.Description' := 'Station ErrorWarning update Enable'}
	DataChangeStatusErrorWarningEnable			: BOOL;

	{attribute 'OPC.UA.DA.Description' := 'Station Current Configuration update Enable'}
	DataChangeStatusCurrentConfigurationEnable	: BOOL;

	{attribute 'OPC.UA.DA.Description' := 'Station Upcoming Configuration update Enable'}
	DataChangeStatusUpcomingConfigurationEnable	: BOOL;

	{attribute 'OPC.UA.DA.Description' := 'Station Operationaldata update Enable'}
	DataChangeStatusOperationalDataEnable		: BOOL;

END_STRUCT
END_TYPE

// ---- ECC/Cell_Unit_4/HeatAndSteam/OPC Data/Sub/AdditionalData/ST_OuputStationHSAdditionalDataOP11600.TcDUT
TYPE ST_OuputStationHSAdditionalDataOP11600 :
STRUCT
	{attribute 'OPC.UA.DA.Description' := 'Dummy (for making struct visible on OPC UA'}
	Dummy						: BOOL;
END_STRUCT
END_TYPE

// ---- ECC/Cell_Unit_4/HeatAndSteam/OPC Data/Sub/AdditionalData/ST_OuputStationHSAdditionalDataOP11601.TcDUT
TYPE ST_OuputStationHSAdditionalDataOP11601 :
STRUCT
	{attribute 'OPC.UA.DA.Description' := 'Dummy (for making struct visible on OPC UA'}
	Dummy						: BOOL;
END_STRUCT
END_TYPE

// ---- ECC/Cell_Unit_4/HeatAndSteam/OPC Data/Sub/Configuration/ST_InputStationHSConfigurationOP11600.TcDUT
TYPE ST_InputStationHSConfigurationOP11600 :
STRUCT
	{attribute 'OPC.UA.DA.Description' := 'Status variables for describing if the operation is restricted for specific SKUs'}
	{attribute 'OPC.UA.DA.StructuredType' := '1'}
	SKURestriction				: ST_SKURestriction;
	
	{attribute 'OPC.UA.DA.Description' := 'Possible tool amount for the operation'}
	ToolCapacity				: UINT;
	
	{attribute 'OPC.UA.DA.Description' := 'Possible material amount for the operation'}
	MaterialCapacity			: UINT;

	{attribute 'OPC.UA.DA.Description' := 'Current config for the operation'}
	{attribute 'OPC.UA.DA.StructuredType' := '1'}
	CurrentConfiguration		: ST_OutputStationHSCurrentConfigurationOP11600;

	{attribute 'OPC.UA.DA.Description' := 'Next config for the operation'}
	{attribute 'OPC.UA.DA.StructuredType' := '1'}
	UpcomingConfiguration		: ST_OutputStationHSUpcomingConfigurationOP11600;

	
END_STRUCT
END_TYPE

// ---- ECC/Cell_Unit_4/HeatAndSteam/OPC Data/Sub/Configuration/ST_InputStationHSUpcomingConfigurationOP11601.TcDUT
TYPE ST_InputStationHSUpcomingConfigurationOP11601 :
STRUCT
	{attribute 'OPC.UA.DA.Description' := 'Number of tools configured for the operation (0-200)'}
	ToolCapacityUsed			: UINT;
	
	{attribute 'OPC.UA.DA.Description' := 'IDs of upcoming tools'}
	{attribute 'OPC.UA.DA.StructuredType' := '1'}
	Tool 						: ARRAY [1..200] OF ToolX;

	{attribute 'OPC.UA.DA.Description' := 'Upcoming number of material configured for the operation (0-200)'}
	MaterialCapacityUsed		: UINT; 

	{attribute 'OPC.UA.DA.Description' := 'IDs OF upcoming material'}
	Material					: ARRAY [1..200] OF STRING(30);

END_STRUCT
END_TYPE

// ---- ECC/Cell_Unit_4/HeatAndSteam/OPC Data/Sub/Configuration/ST_InputStationHSConfigurationOP11601.TcDUT
TYPE ST_InputStationHSConfigurationOP11601 :
STRUCT
	{attribute 'OPC.UA.DA.Description' := 'Status variables for describing if the operation is restricted for specific SKUs'}
	{attribute 'OPC.UA.DA.StructuredType' := '1'}
	SKURestriction				: ST_SKURestriction;
	
	{attribute 'OPC.UA.DA.Description' := 'Possible tool amount for the operation'}
	ToolCapacity				: UINT;
	
	{attribute 'OPC.UA.DA.Description' := 'Possible material amount for the operation'}
	MaterialCapacity			: UINT;

	{attribute 'OPC.UA.DA.Description' := 'Current config for the operation'}
	{attribute 'OPC.UA.DA.StructuredType' := '1'}
	CurrentConfiguration		: ST_OutputStationHSCurrentConfigurationOP11601;

	{attribute 'OPC.UA.DA.Description' := 'Next config for the operation'}
	{attribute 'OPC.UA.DA.StructuredType' := '1'}
	UpcomingConfiguration		: ST_OutputStationHSUpcomingConfigurationOP11601;

	
END_STRUCT
END_TYPE

// ---- ECC/Cell_Unit_4/HeatAndSteam/OPC Data/Sub/Configuration/ST_OutputStationHSCurrentConfigurationOP11601.TcDUT
TYPE ST_OutputStationHSCurrentConfigurationOP11601 :
STRUCT
	{attribute 'OPC.UA.DA.Description' := 'Status variables for describing if the operation is restricted for specific SKUs'}
	{attribute 'OPC.UA.DA.StructuredType' := '1'}
	SKURestriction				: ST_SKURestriction;
	
	{attribute 'OPC.UA.DA.Description' := 'Possible tool amount for the operation'}
	ToolCapacity				: UINT;
	
	{attribute 'OPC.UA.DA.Description' := 'Number of tools configured for the operation (0-200)'}
	ToolCapacityUsed			: UINT;

	{attribute 'OPC.UA.DA.Description' := 'IDs of upcoming tools'}
	{attribute 'OPC.UA.DA.StructuredType' := '1'}
	Tool 						: ARRAY [1..200] OF ToolX;

	{attribute 'OPC.UA.DA.Description' := 'Status variables for current location and control mapping of tools'}
	{attribute 'OPC.UA.DA.StructuredType' := '1'}
	ToolMapping					: ARRAY [1..200] OF ToolXMapping;

	{attribute 'OPC.UA.DA.Description' := 'Possible material amount for the operation'}
	MaterialCapacity			: UINT;
	
	{attribute 'OPC.UA.DA.Description' := 'Upcoming number of material configured for the operation (0-200)'}
	MaterialCapacityUsed		: UINT; 

	{attribute 'OPC.UA.DA.Description' := 'IDs OF upcoming material'}
	Material					: ARRAY [1..200] OF STRING(30);

	{attribute 'OPC.UA.DA.Description' := 'Status variables for current location and control mapping of feeding material'}
	{attribute 'OPC.UA.DA.StructuredType' := '1'}
	MaterialMapping				: ARRAY [1..200] OF MaterialXMapping;
END_STRUCT
END_TYPE

// ---- ECC/Cell_Unit_4/HeatAndSteam/OPC Data/Sub/Configuration/ST_OutputStationHSUpcomingConfigurationOP11601.TcDUT
TYPE ST_OutputStationHSUpcomingConfigurationOP11601 :
STRUCT
	{attribute 'OPC.UA.DA.Description' := 'Number of tools configured for the operation (0-200)'}
	ToolCapacityUsed			: UINT;

	{attribute 'OPC.UA.DA.Description' := 'IDs of upcoming tools'}
	{attribute 'OPC.UA.DA.StructuredType' := '1'}
	Tool 						: ARRAY [1..200] OF ToolX;

	{attribute 'OPC.UA.DA.Description' := 'Upcoming number of material configured for the operation (0-200)'}
	MaterialCapacityUsed		: UINT; 

	{attribute 'OPC.UA.DA.Description' := 'IDs OF upcoming material'}
	Material					: ARRAY [1..200] OF STRING(30);

END_STRUCT
END_TYPE

// ---- ECC/Cell_Unit_4/HeatAndSteam/OPC Data/Sub/Control/ST_InputStationHSControlOP11601.TcDUT
TYPE ST_InputStationHSControlOP11601 :
STRUCT
	{attribute 'OPC.UA.DA.Description' := 'Dummy (for making struct visible on OPC UA'}
	Dummy						: BOOL;
END_STRUCT
END_TYPE

// ---- ECC/Cell_Unit_4/HeatAndSteam/OPC Data/Sub/JobData/ST_OutputStationHSJobDataOP11600.TcDUT
TYPE ST_OutputStationHSJobDataOP11600 :
STRUCT
	{attribute 'OPC.UA.DA.Description' := 'Dynamic Tool'}
	{attribute 'OPC.UA.DA.StructuredType' := '1'}
	DynamicTool						: ARRAY [1..1] OF ToolX;

	{attribute 'OPC.UA.DA.Description' := 'Dynamic Material'}
	DynamicMaterial					: ARRAY [1..1] OF STRING(30);

	{attribute 'OPC.UA.DA.Description' := 'Temperature Target C°'}
	TemperatureTarget				: REAL;

	{attribute 'OPC.UA.DA.Description' := 'Temperature Max C°'}
	TemperatureMax					: REAL;
	
	{attribute 'OPC.UA.DA.Description' := 'Temperature Min C°'}
	TemperatureMin					: REAL;
	
	{attribute 'OPC.UA.DA.Description' := 'Time Max S'}
	TimeMax							: REAL;
	
	{attribute 'OPC.UA.DA.Description' := 'Time Min S'}
	TimeMin							: REAL;
	
	{attribute 'OPC.UA.DA.Description' := 'Steam Max'}
	SteamMax						: REAL;
	
	{attribute 'OPC.UA.DA.Description' := 'Steam Min'}
	SteamMin						: REAL;
	
	{attribute 'OPC.UA.DA.Description' := 'Air Max'}
	AirMax							: REAL;
	
	{attribute 'OPC.UA.DA.Description' := 'Air Min'}
	AirMin							: REAL;
	
	{attribute 'OPC.UA.DA.Description' := 'Profile'}
	Profile							: ARRAY [ 1..10] OF REAL;
	
END_STRUCT
END_TYPE

// ---- ECC/Cell_Unit_4/HeatAndSteam/OPC Data/Sub/JobData/ST_InputStationHSJobDataOP11601.TcDUT
TYPE ST_InputStationHSJobDataOP11601 :
STRUCT
	{attribute 'OPC.UA.DA.Description' := 'Dynamic Tool'}
	{attribute 'OPC.UA.DA.StructuredType' := '1'}
	DynamicTool						: ARRAY [1..1] OF ToolX;

	{attribute 'OPC.UA.DA.Description' := 'Dynamic Material'}
	DynamicMaterial					: ARRAY [1..1] OF STRING(30);

	{attribute 'OPC.UA.DA.Description' := 'Temperature Target C°'}
	TemperatureTarget				: REAL;

	{attribute 'OPC.UA.DA.Description' := 'Temperature Max C°'}
	TemperatureMax					: REAL;
	
	{attribute 'OPC.UA.DA.Description' := 'Temperature Min C°'}
	TemperatureMin					: REAL;
	
	{attribute 'OPC.UA.DA.Description' := 'Time Max S'}
	TimeMax							: REAL;
	
	{attribute 'OPC.UA.DA.Description' := 'Time Min S'}
	TimeMin							: REAL;
	
	{attribute 'OPC.UA.DA.Description' := 'Steam Max'}
	SteamMax						: REAL;
	
	{attribute 'OPC.UA.DA.Description' := 'Steam Min'}
	SteamMin						: REAL;
	
	{attribute 'OPC.UA.DA.Description' := 'Air Max'}
	AirMax							: REAL;
	
	{attribute 'OPC.UA.DA.Description' := 'Air Min'}
	AirMin							: REAL;
	
	{attribute 'OPC.UA.DA.Description' := 'Profile'}
	Profile							: ARRAY [ 1..10] OF REAL;

END_STRUCT
END_TYPE

// ---- ECC/Cell_Unit_4/HeatAndSteam/OPC Data/Sub/JobData/ST_OutputStationHSJobDataOP11601.TcDUT
TYPE ST_OutputStationHSJobDataOP11601 :
STRUCT
	{attribute 'OPC.UA.DA.Description' := 'Dynamic Tool'}
	{attribute 'OPC.UA.DA.StructuredType' := '1'}
	DynamicTool						: ARRAY [1..1] OF ToolX;

	{attribute 'OPC.UA.DA.Description' := 'Dynamic Material'}
	DynamicMaterial					: ARRAY [1..1] OF STRING(30);

	{attribute 'OPC.UA.DA.Description' := 'Temperature Target C°'}
	TemperatureTarget				: REAL;

	{attribute 'OPC.UA.DA.Description' := 'Temperature Max C°'}
	TemperatureMax					: REAL;
	
	{attribute 'OPC.UA.DA.Description' := 'Temperature Min C°'}
	TemperatureMin					: REAL;
	
	{attribute 'OPC.UA.DA.Description' := 'Time Max S'}
	TimeMax							: REAL;
	
	{attribute 'OPC.UA.DA.Description' := 'Time Min S'}
	TimeMin							: REAL;
	
	{attribute 'OPC.UA.DA.Description' := 'Steam Max'}
	SteamMax						: REAL;
	
	{attribute 'OPC.UA.DA.Description' := 'Steam Min'}
	SteamMin						: REAL;
	
	{attribute 'OPC.UA.DA.Description' := 'Air Max'}
	AirMax							: REAL;
	
	{attribute 'OPC.UA.DA.Description' := 'Air Min'}
	AirMin							: REAL;
	
	{attribute 'OPC.UA.DA.Description' := 'Profile'}
	Profile							: ARRAY [ 1..10] OF REAL;
	
END_STRUCT
END_TYPE

// ---- ECC/Cell_Unit_4/HeatAndSteam/OPC Data/Sub/OperationalData/ST_OutputStationHSOperationalDataOP11601.TcDUT
TYPE ST_OutputStationHSOperationalDataOP11601 :
STRUCT
	{attribute 'OPC.UA.DA.Description' := 'Current number of tools where data is available'}
	NumberOfToolData			: UINT;

	{attribute 'OPC.UA.DA.Description' := 'Status variables for current operational data of tools'}
	{attribute 'OPC.UA.DA.StructuredType' := '1'}
	ToolData					: ARRAY [1..200] OF ToolDataX;

	{attribute 'OPC.UA.DA.Description' := 'Current number OF feeding material where data is available'}
	NumberOfMaterialData		: UINT;

	{attribute 'OPC.UA.DA.Description' := 'Status variables for current operational data of material'}
	{attribute 'OPC.UA.DA.StructuredType' := '1'}
	MaterialData				: ARRAY [1..200] OF MaterialDataX;

//	{attribute 'OPC.UA.DA.Description' := 'Status variables FOR current operational data of devices'}
//	{attribute 'OPC.UA.DA.StructuredType' := '1'}
//	DeviceData					: ST_Scanner_JobStatus;
	
END_STRUCT
END_TYPE

// ---- ECC/Cell_Unit_4/HeatAndSteam/stStationVehicleCmdOut.TcDUT
TYPE stStationVehicleCmdOut :
STRUCT
	bCmdStart			: BOOL;
	iVehicleID			: UINT;
	iBufferDestination 	: UINT;
	iVehilceVelocity	: REAL;
END_STRUCT
END_TYPE

// ---- ECC/Cell_Unit_4/OPC Data/ST_Input.TcDUT
/// Specialized Bridge input for SOR cell
TYPE ST_Input :
STRUCT
	{attribute 'OPC.UA.DA.Description' := 'Bridge header'}
	{attribute 'OPC.UA.DA.StructuredType' := '1'}
	{attribute 'TcIgnorePersistent'}
	Header					: ST_InputHeader;

	{attribute 'OPC.UA.DA.Description' := 'Bridge Cell Data'}
	{attribute 'OPC.UA.DA.StructuredType' := '1'}
	Cell					: ST_InputCell;

	{attribute 'OPC.UA.DA.Description' := 'Bridge Station Data'}
	{attribute 'OPC.UA.DA.StructuredType' := '1'}
	Station					: ST_InputStation;

	{attribute 'OPC.UA.DA.Description' := 'Bridge additional data'}
	{attribute 'OPC.UA.DA.StructuredType' := '1'}
	Transport				: ST_InputTransport;

END_STRUCT
END_TYPE

// ---- ECC/Cell_Unit_4/OPC Data/ST_Output.TcDUT
TYPE ST_Output :
STRUCT
	{attribute 'OPC.UA.DA.Description' := 'Bridge header'}
	{attribute 'OPC.UA.DA.StructuredType' := '1'}
	{attribute 'TcIgnorePersistent'}
	Header					: ST_OutputHeader;
	
	{attribute 'OPC.UA.DA.Description' := 'Bridge Cell Data'}
	{attribute 'OPC.UA.DA.StructuredType' := '1'}
	Cell					: ST_OutputCell;

	{attribute 'OPC.UA.DA.Description' := 'Bridge Station 1 Data'}
	{attribute 'OPC.UA.DA.StructuredType' := '1'}
	Station					: ST_OutputStation;
	
	{attribute 'OPC.UA.DA.Description' := 'Bridge transport data'}
	{attribute 'OPC.UA.DA.StructuredType' := '1'}
	Transport				: ST_OutputTransport;

END_STRUCT
END_TYPE

// ---- ECC/Cell_Unit_4/OPC Data/Sub/ST_InputCell.TcDUT
TYPE ST_InputCell :
STRUCT
	{attribute 'OPC.UA.DA.Description' := 'Cell Mode State'}
	{attribute 'OPC.UA.DA.StructuredType' := '1'}
	{attribute 'TcIgnorePersistent'}
	ModeState			: ST_InputModeState;

	{attribute 'OPC.UA.DA.Description' := 'Cell Configuration'}
	{attribute 'OPC.UA.DA.StructuredType' := '1'}
	Configuration		: ST_InputCellConfiguration;
	
	{attribute 'OPC.UA.DA.Description' := 'Cell Control'}
	{attribute 'OPC.UA.DA.StructuredType' := '1'}
	{attribute 'TcIgnorePersistent'}
	Control				: ST_InputCellControl;

	{attribute 'OPC.UA.DA.Description' := 'Cell Additional Data'}
	{attribute 'OPC.UA.DA.StructuredType' := '1'}
	{attribute 'TcIgnorePersistent'}
	AdditionalData		: ST_InputCellAdditionalData;

END_STRUCT
END_TYPE

// ---- ECC/Cell_Unit_4/OPC Data/Sub/ST_InputCellAdditionalData.TcDUT
/// Standard Additional Data for cells
TYPE ST_InputCellAdditionalData :
STRUCT
	{attribute 'OPC.UA.DA.Description' := 'Cell MES Handshakes'}
	{attribute 'OPC.UA.DA.StructuredType' := '1'}
	{attribute 'TcIgnorePersistent'}
	MESHandShakes				: ST_InputCellAdditionalDataMESHandShake;

	{attribute 'OPC.UA.DA.Description' := 'Cell MES Handshakes'}
	{attribute 'OPC.UA.DA.StructuredType' := '1'}
	Settings					: ST_InputCellAdditionalDataSettings;
	
	{attribute 'OPC.UA.DA.Description' := 'Clear all ticket data on cell'}
	ClearAll					: BOOL;			
	
END_STRUCT
END_TYPE

// ---- ECC/Cell_Unit_4/OPC Data/Sub/ST_InputCellAdditionalDataMESHandShake.TcDUT
TYPE ST_InputCellAdditionalDataMESHandShake :
STRUCT
	{attribute 'OPC.UA.DA.Description' := 'Cell ModeState update status'}
	{attribute 'TcIgnorePersistent'}
	DataChangeStatusModeState		: UINT;

	{attribute 'OPC.UA.DA.Description' := 'Cell OEE update status'}
	{attribute 'TcIgnorePersistent'}
	DataChangeStatusOEE				: UINT;

	{attribute 'OPC.UA.DA.Description' := 'Cell ErrorWarning update status'}
	{attribute 'TcIgnorePersistent'}
	DataChangeStatusErrorWarning	: UINT;

	{attribute 'OPC.UA.DA.Description' := 'Cell Operationaldata update status'}
	{attribute 'TcIgnorePersistent'}
	DataChangeStatusOperationalData	: UINT;

END_STRUCT
END_TYPE

// ---- ECC/Cell_Unit_4/OPC Data/Sub/ST_InputCellAdditionalDataSettings.TcDUT
TYPE ST_InputCellAdditionalDataSettings :
STRUCT
	{attribute 'OPC.UA.DA.Description' := 'Cell ModeState update Enable'}
	DataChangeStatusModeStateEnable			: BOOL;

	{attribute 'OPC.UA.DA.Description' := 'Cell OEE update Enable'}
	DataChangeStatusOEEEnable				: BOOL;

	{attribute 'OPC.UA.DA.Description' := 'Cell ErrorWarning update Enable'}
	DataChangeStatusErrorWarningEnable		: BOOL;

	{attribute 'OPC.UA.DA.Description' := 'Cell Operationaldata update Enable'}
	DataChangeStatusOperationalDataEnable	: BOOL;

END_STRUCT
END_TYPE

// ---- ECC/Cell_Unit_4/OPC Data/Sub/ST_InputCellConfiguration.TcDUT
/// Specialized Config for SOR cell
TYPE ST_InputCellConfiguration :
STRUCT
	{attribute 'OPC.UA.DA.Description' := 'Change Request (0-255)'}
	ChangeRequest				: UINT;

	{attribute 'OPC.UA.DA.Description' := 'Cell general configuration'}
	{attribute 'OPC.UA.DA.StructuredType' := '1'}
	General						: ST_InputCellConfigurationGeneral;

END_STRUCT
END_TYPE

// ---- ECC/Cell_Unit_4/OPC Data/Sub/ST_InputCellConfigurationGeneral.TcDUT
/// Specialized Config for SOR cell
TYPE ST_InputCellConfigurationGeneral :
STRUCT
	{attribute 'OPC.UA.DA.Description' := 'Dummy (for making struct visible on OPC UA'}
	Dummy						: BOOL;

END_STRUCT
END_TYPE

// ---- ECC/Cell_Unit_4/OPC Data/Sub/ST_InputCellControl.TcDUT
TYPE ST_InputCellControl :
STRUCT
	{attribute 'OPC.UA.DA.Description' := 'Reset E-Stop'}
	ResetEStop					: BOOL;

	{attribute 'OPC.UA.DA.Description' := 'Lock cell doors'}
	LockDoors					: BOOL;

	{attribute 'OPC.UA.DA.Description' := 'Unlock cell doors'}
	UnlockDoors					: BOOL;

	{attribute 'OPC.UA.DA.Description' := 'Turn on cell lights'}
	EnableCellLight				: BOOL;

END_STRUCT
END_TYPE

// ---- ECC/Cell_Unit_4/OPC Data/Sub/ST_InputStation.TcDUT
TYPE ST_InputStation :
STRUCT
	{attribute 'OPC.UA.DA.Description' := 'Bridge Station 1 Data'}
	{attribute 'OPC.UA.DA.StructuredType' := '1'}
	Station1			: ST_InputStationStationHS;
	{attribute 'OPC.UA.DA.Description' := 'Bridge Station 2 Data'}
	{attribute 'OPC.UA.DA.StructuredType' := '1'}
	Station2			: ST_InputStationStationHS;
END_STRUCT
END_TYPE

// ---- ECC/Cell_Unit_4/OPC Data/Sub/ST_OutputCell.TcDUT
TYPE ST_OutputCell :
STRUCT
	{attribute 'OPC.UA.DA.Description' := 'Cell Mode State'}
	{attribute 'OPC.UA.DA.StructuredType' := '1'}
	ModeState			: ST_OutputModeState;

	{attribute 'OPC.UA.DA.Description' := 'Cell OEE'}
	{attribute 'OPC.UA.DA.StructuredType' := '1'}
	OEE					: ST_OutputOEE;
	
	{attribute 'OPC.UA.DA.Description' := 'Cell error warning'}
	{attribute 'OPC.UA.DA.StructuredType' := '1'}
	ErrorWarning		: ST_OutputErrorWarning;
	
	{attribute 'OPC.UA.DA.Description' := 'Cell configuration'}
	{attribute 'OPC.UA.DA.StructuredType' := '1'}
	Configuration		: ST_OutputCellConfiguration;
	
	{attribute 'OPC.UA.DA.Description' := 'Cell operational data'}
	{attribute 'OPC.UA.DA.StructuredType' := '1'}
	OperationalData		: ST_OutputCellOperationalData;

	{attribute 'OPC.UA.DA.Description' := 'Cell operational data'}
	{attribute 'OPC.UA.DA.StructuredType' := '1'}
	SustainabilityData	: ST_OutputCellSustainabilityData;

	{attribute 'OPC.UA.DA.Description' := 'Cell additional data'}
	{attribute 'OPC.UA.DA.StructuredType' := '1'}
	AdditionalData		: ST_OutputCellAdditionalData;

END_STRUCT
END_TYPE

// ---- ECC/Cell_Unit_4/OPC Data/Sub/ST_OutputCellAdditionalData.TcDUT
TYPE ST_OutputCellAdditionalData :
STRUCT
	{attribute 'OPC.UA.DA.Description' := 'Dummy (for making struct visible on OPC UA'}
	Dummy						: BOOL;

END_STRUCT
END_TYPE

// ---- ECC/Cell_Unit_4/OPC Data/Sub/ST_OutputCellConfiguration.TcDUT
TYPE ST_OutputCellConfiguration :
STRUCT
// Handshake part
	{attribute 'OPC.UA.DA.Description' := 'Change acknowledge (0-255)'}
	ChangeAcknowledge				: UINT;

	{attribute 'OPC.UA.DA.Description' := 'Change status (0-255)'}
	ChangeStatus					: UINT;

// Data part
	{attribute 'OPC.UA.DA.Description' := 'Data Changed (0-65536)'}
	DataChange						: UINT;

	{attribute 'OPC.UA.DA.Description' := 'Data Changed (0-65536)'}
	{attribute 'OPC.UA.DA.StructuredType' := '1'}
	General							: ST_OutputCellConfigurationGeneral;
	
END_STRUCT
END_TYPE

// ---- ECC/Cell_Unit_4/OPC Data/Sub/ST_OutputCellConfigurationGeneral.TcDUT
/// Specialized Config for SOR cell
TYPE ST_OutputCellConfigurationGeneral :
STRUCT
	{attribute 'OPC.UA.DA.Description' := 'Dummy (for making struct visible on OPC UA'}
	Dummy						: BOOL;

END_STRUCT
END_TYPE

// ---- ECC/Cell_Unit_4/OPC Data/Sub/ST_OutputCellOperationalData.TcDUT
TYPE ST_OutputCellOperationalData :
STRUCT
// Handshake part
	{attribute 'OPC.UA.DA.Description' := 'Change acknowledged (0-255)'}
	ChangeAcknowledge			: UINT;

	{attribute 'OPC.UA.DA.Description' := 'Change status (0-255)'}
	ChangeStatus				: UINT;

// Data part	
	{attribute 'OPC.UA.DA.Description' := 'Data has changed (0-65536)'}
	DataChange					: UINT;

	{attribute 'OPC.UA.DA.Description' := 'General'}
	{attribute 'OPC.UA.DA.StructuredType' := '1'}
	General						: ST_OutputCellOperationalDataGeneral;
	
	{attribute 'OPC.UA.DA.Description' := 'Status variables for current operational data of devices'}
	{attribute 'OPC.UA.DA.StructuredType' := '1'}
	DeviceData					: ARRAY [1..200] OF ST_DeviceDataX;
	
END_STRUCT
END_TYPE

// ---- ECC/Cell_Unit_4/OPC Data/Sub/ST_OutputCellSustainabilityData.TcDUT
TYPE ST_OutputCellSustainabilityData :
STRUCT
	// Handshake part
	{attribute 'OPC.UA.DA.Description' := 'Change acknowledged (0-255)'}
	ChangeAcknowledge			: UINT;

	{attribute 'OPC.UA.DA.Description' := 'Change status (0-255)'}
	ChangeStatus				: UINT;

	// Data part	
	{attribute 'OPC.UA.DA.Description' := 'Data has changed (0-65536)'}
	DataChange					: UINT;
	
	{attribute 'OPC.UA.DA.Description' := 'Status variables for current sustainability data of devices'}
	{attribute 'OPC.UA.DA.StructuredType' := '1'}
	Energy						: ARRAY [1..200] OF ST_DeviceDataX;
	
	{attribute 'OPC.UA.DA.Description' := 'Status variables for current sustainability data of devices'}
	{attribute 'OPC.UA.DA.StructuredType' := '1'}
	Fluid						: ARRAY [1..200] OF ST_DeviceDataX;
	
	{attribute 'OPC.UA.DA.Description' := 'Status variables for current sustainability data of devices'}
	{attribute 'OPC.UA.DA.StructuredType' := '1'}
	Exhaust						: ARRAY [1..200] OF ST_DeviceDataX;

END_STRUCT
END_TYPE

// ---- ECC/Cell_Unit_4/OPC Data/Sub/ST_OutputHeader.TcDUT
TYPE ST_OutputHeader :
STRUCT
	{attribute 'OPC.UA.DA.Description' := 'Header (0-100, 2 Hz)'}
	HeartBeat				: UINT;

	{attribute 'OPC.UA.DA.Description' := 'Cell information'}
	{attribute 'OPC.UA.DA.StructuredType' := '1'}
	CellInformation			: ST_OutputHeaderCellInformation;
	
	{attribute 'OPC.UA.DA.Description' := 'Cell information'}
	{attribute 'OPC.UA.DA.StructuredType' := '1'}
	MetaInformation			: ST_OutputHeaderMetaInformationX;
	
END_STRUCT
END_TYPE

// ---- ECC/Cell_Unit_4/OPC Data/Sub/ST_OutputHeaderCellInformation.TcDUT
TYPE ST_OutputHeaderCellInformation:// EXTENDS ST_OutputHeaderCellInformationX :
STRUCT
	{attribute 'OPC.UA.DA.Description' := 'Station information'}
	{attribute 'OPC.UA.DA.StructuredType' := '1'}
	StationInformation		: ARRAY [1..2] OF ST_OutputHeaderCellInformationStationHS;
	
	{attribute 'OPC.UA.DA.Description' := 'Cell name'}
	CellName				: STRING;

	{attribute 'OPC.UA.DA.Description' := 'CellID'}
	CellID					: STRING;

	{attribute 'OPC.UA.DA.Description' := 'Number of stations'}
	NumberOfStations		: UINT;

	{attribute 'OPC.UA.DA.Description' := 'Station information'}
	{attribute 'OPC.UA.DA.StructuredType' := '1'}
	TransportInformation	: ST_OutputHeaderTransportInformationX;

END_STRUCT
END_TYPE

// ---- ECC/Cell_Unit_4/OPC Data/Sub/ST_OutputHeaderCellInformationStation.TcDUT
TYPE ST_OutputHeaderCellInformationStation :
STRUCT
	StationInformation			: ARRAY [1..2] OF ST_OutputHeaderCellInformationStationHS;
END_STRUCT
END_TYPE

// ---- ECC/Cell_Unit_4/OPC Data/Sub/ST_OutputHeaderCellInformationStationInformationOperationInformation.TcDUT
TYPE ST_OutputHeaderCellInformationStationInformationOperationInformation :
STRUCT
	{attribute 'OPC.UA.DA.Description' := 'Operation information'}
	{attribute 'OPC.UA.DA.StructuredType' := '1'}
	OperationInformation		: ARRAY [1..4] OF ST_OutputHeaderCellInformationStationInformationOperationInformationX;
END_STRUCT
END_TYPE

// ---- ECC/Cell_Unit_4/OPC Data/Sub/ST_OutputStation.TcDUT
TYPE ST_OutputStation :
STRUCT
	{attribute 'OPC.UA.DA.Description' := 'Bridge Station 1 Data'}
	{attribute 'OPC.UA.DA.StructuredType' := '1'}
	Station1			: ST_OutputStationStationHS;
		{attribute 'OPC.UA.DA.Description' := 'Bridge Station 2 Data'}
	{attribute 'OPC.UA.DA.StructuredType' := '1'}
	Station2			: ST_OutputStationStationHS;
END_STRUCT
END_TYPE

// ---- ECC/Cell_Unit_4/HeatAndSteam/E_HSStationINSeq.TcDUT
{attribute 'qualified_only'}
{attribute 'strict'}
TYPE E_HSStationINSeq :
(
	Idle := 0,
	NewJob,
	CheckVehiclesVelocity,
	CheckVehiclesSettings,
	SetSettingsOnDevice,
	WaitForDeviceReady,
	ReceiveNextVehicle,
	Running,
	WaitBeforeEmpty,
	Done
);
END_TYPE

// ---- ECC/Cell_Unit_4/HeatAndSteam/OPC Data/ST_InputStationStationHS.TcDUT
TYPE ST_InputStationStationHS :
STRUCT
	{attribute 'OPC.UA.DA.Description' := 'Station mode and state'}
	{attribute 'OPC.UA.DA.StructuredType' := '1'}
	{attribute 'TcIgnorePersistent'}
	ModeState			: ST_InputModeState;

	{attribute 'OPC.UA.DA.Description' := 'Station job data'}
	{attribute 'OPC.UA.DA.StructuredType' := '1'}
	JobData				: ST_InputStationHSJobData;

	{attribute 'OPC.UA.DA.Description' := 'Station configuration'}
	{attribute 'OPC.UA.DA.StructuredType' := '1'}
	CurrentConfiguration: ST_InputStationHSConfiguration;

	{attribute 'OPC.UA.DA.Description' := 'Station configuration'}
	{attribute 'OPC.UA.DA.StructuredType' := '1'}
	UpcomingConfiguration: ST_InputStationHSUpcomingConfiguration;

	{attribute 'OPC.UA.DA.Description' := 'Station configuration'}
	{attribute 'OPC.UA.DA.StructuredType' := '1'}
	Control				: ST_InputStationHSControl;

	{attribute 'OPC.UA.DA.Description' := 'Station configuration'}
	{attribute 'OPC.UA.DA.StructuredType' := '1'}
	AdditionalData		: ST_InputStationHSAdditionalData;

END_STRUCT
END_TYPE

// ---- ECC/Cell_Unit_4/HeatAndSteam/OPC Data/ST_OutputStationStationHS.TcDUT
TYPE ST_OutputStationStationHS :
STRUCT
		{attribute 'OPC.UA.DA.Description' := 'Station mode and state'}
	{attribute 'OPC.UA.DA.StructuredType' := '1'}
	ModeState			: ST_OutputModeState;
	
	{attribute 'OPC.UA.DA.Description' := 'Station job data'}
	{attribute 'OPC.UA.DA.StructuredType' := '1'}
	JobData				: ST_OutputStationHSJobData;

	{attribute 'OPC.UA.DA.Description' := 'Station OEE'}
	{attribute 'OPC.UA.DA.StructuredType' := '1'}
	OEE					: ST_OutputOEE;

	{attribute 'OPC.UA.DA.Description' := 'Station error/warning'}
	{attribute 'OPC.UA.DA.StructuredType' := '1'}
	ErrorWarning		: ST_OutputErrorWarning;

	{attribute 'OPC.UA.DA.Description' := 'Station configuration'}
	{attribute 'OPC.UA.DA.StructuredType' := '1'}
	CurrentConfiguration: ST_OutputStationHSCurrentConfiguration;

	{attribute 'OPC.UA.DA.Description' := 'Station configuration'}
	{attribute 'OPC.UA.DA.StructuredType' := '1'}
	UpcomingConfiguration: ST_OutputStationHSUpcomingConfiguration;

	{attribute 'OPC.UA.DA.Description' := 'Station operational data'}
	{attribute 'OPC.UA.DA.StructuredType' := '1'}
	OperationalData		: ST_OutputStationHSOperationalData;

	{attribute 'OPC.UA.DA.Description' := 'Station sustainability data'}
	{attribute 'OPC.UA.DA.StructuredType' := '1'}
	SustainabilityData	: ST_OutputStationHSSustainabilityData;

	{attribute 'OPC.UA.DA.Description' := 'Station sustainability data'}
	{attribute 'OPC.UA.DA.StructuredType' := '1'}
	AdditionalData		: ST_OutputStationHSAdditionalData;
END_STRUCT
END_TYPE

// ---- ECC/Cell_Unit_4/HeatAndSteam/OPC Data/Sub/AdditionalData/ST_InputStationHSAdditionalData.TcDUT
TYPE ST_InputStationHSAdditionalData :
STRUCT
	{attribute 'OPC.UA.DA.Description' := 'Station MES Handshakes'}
	{attribute 'OPC.UA.DA.StructuredType' := '1'}
	{attribute 'TcIgnorePersistent'}
	MESHandShakes				: ST_InputStationHSAdditionalDataMESHandShake;

	{attribute 'OPC.UA.DA.Description' := 'Cell MES Handshakes'}
	{attribute 'OPC.UA.DA.StructuredType' := '1'}
	Settings					: ST_InputStationHSAdditionalDataSettings;
	
	{attribute 'OPC.UA.DA.Description' := 'Station general additional data'}
	{attribute 'OPC.UA.DA.StructuredType' := '1'}
	General						: ST_InputStationHSAdditionalDataGeneral;
	
	(* Might not be the same struct *)
	{attribute 'OPC.UA.DA.Description' := 'HeatAndSteam Step 1 additional data'}
	{attribute 'OPC.UA.DA.StructuredType' := '1'}
	OP11600						: ST_InputStationHSAdditionalDataOP11600;

//	{attribute 'OPC.UA.DA.Description' := 'HeatAndSteam Step 2 additional data'}
//	{attribute 'OPC.UA.DA.StructuredType' := '1'}
//	OP11601						: ST_InputStationHSAdditionalDataOP11601;
END_STRUCT
END_TYPE

// ---- ECC/Cell_Unit_4/HeatAndSteam/OPC Data/Sub/AdditionalData/ST_InputStationHSAdditionalDataGeneral.TcDUT
TYPE ST_InputStationHSAdditionalDataGeneral :
STRUCT
	{attribute 'OPC.UA.DA.Description' := 'Dummy (for making struct visible on OPC UA'}
	{attribute 'TcIgnorePersistent'}
	Dummy						: BOOL;
END_STRUCT
END_TYPE

// ---- ECC/Cell_Unit_4/HeatAndSteam/OPC Data/Sub/AdditionalData/ST_OutputStationHSAdditionalData.TcDUT
TYPE ST_OutputStationHSAdditionalData :
STRUCT
	{attribute 'OPC.UA.DA.Description' := 'General'}
	{attribute 'OPC.UA.DA.StructuredType' := '1'}
	General					: ST_OutputStationHSAdditionalDataGeneral;

	(* Might not be the same struct *)
	{attribute 'OPC.UA.DA.Description' := 'HeatAndSteam Step 1 additional data'}
	{attribute 'OPC.UA.DA.StructuredType' := '1'}
	OP11600					: ST_OuputStationHSAdditionalDataOP11600;

//	{attribute 'OPC.UA.DA.Description' := 'HeatAndSteam Step 2 additional data'}
//	{attribute 'OPC.UA.DA.StructuredType' := '1'}
//	OP11601					: ST_OuputStationHSAdditionalDataOP11601;
END_STRUCT
END_TYPE

// ---- ECC/Cell_Unit_4/HeatAndSteam/OPC Data/Sub/AdditionalData/ST_OutputStationHSAdditionalDataGeneral.TcDUT
TYPE ST_OutputStationHSAdditionalDataGeneral :
STRUCT
	{attribute 'OPC.UA.DA.Description' := 'Dummy (for making struct visible on OPC UA'}
	Dummy						: BOOL;
END_STRUCT
END_TYPE

// ---- ECC/Cell_Unit_4/HeatAndSteam/OPC Data/Sub/Configuration/ST_InputStationHSConfiguration.TcDUT
TYPE ST_InputStationHSConfiguration :
STRUCT
	{attribute 'OPC.UA.DA.Description' := 'Change Request (0-255)'}
	{attribute 'TcIgnorePersistent'}
	ChangeRequest				: UINT;
	
	{attribute 'OPC.UA.DA.Description' := 'Configuration type (OPxxxxx or General)'}
	{attribute 'TcIgnorePersistent'}
	ConfigurationType			: STRING(7);
	
	{attribute 'OPC.UA.DA.Description' := 'Station general configuration'}
	{attribute 'OPC.UA.DA.StructuredType' := '1'}
	General						: ST_InputStationHSConfigurationGeneral;
	
		(* Might not be the same struct *)
	{attribute 'OPC.UA.DA.Description' := 'HeatAndSteam Step 1 Configuration'}
	{attribute 'OPC.UA.DA.StructuredType' := '1'}
	OP11600						: ST_InputStationHSConfigurationOP11600;

//	{attribute 'OPC.UA.DA.Description' := 'HeatAndSteam Step 2 Configuration'}
//	{attribute 'OPC.UA.DA.StructuredType' := '1'}
//	OP11601						: ST_InputStationHSConfigurationOP11601;

END_STRUCT
END_TYPE

// ---- ECC/Cell_Unit_4/HeatAndSteam/OPC Data/Sub/Configuration/ST_InputStationHSConfigurationGeneral.TcDUT
TYPE ST_InputStationHSConfigurationGeneral :
STRUCT
	{attribute 'OPC.UA.DA.Description' := 'Dummy (for making struct visible on OPC UA'}
	Dummy						: BOOL;
END_STRUCT
END_TYPE

// ---- ECC/Cell_Unit_4/HeatAndSteam/OPC Data/Sub/Configuration/ST_InputStationHSUpcomingConfiguration.TcDUT
TYPE ST_InputStationHSUpcomingConfiguration :
STRUCT
	{attribute 'OPC.UA.DA.Description' := 'Change Request (0-255)'}
	{attribute 'TcIgnorePersistent'}
	ChangeRequest				: UINT;
	
	{attribute 'OPC.UA.DA.Description' := 'Configuration type (OPxxxxx or General)'}
	{attribute 'TcIgnorePersistent'}
	ConfigurationType			: STRING(7);
	
	{attribute 'OPC.UA.DA.Description' := 'HeatAndSteam Step 1 Configuration'}
	{attribute 'OPC.UA.DA.StructuredType' := '1'}
	OP11600						: ST_InputStationHSUpcomingConfigurationOP11600;

//	{attribute 'OPC.UA.DA.Description' := 'HeatAndSteam Step 2 Configuration'}
//	{attribute 'OPC.UA.DA.StructuredType' := '1'}
//	OP11601						: ST_InputStationHSUpcomingConfigurationOP11601;
	
END_STRUCT
END_TYPE

// ---- ECC/Cell_Unit_4/HeatAndSteam/OPC Data/Sub/Configuration/ST_InputStationHSUpcomingConfigurationOP11600.TcDUT
TYPE ST_InputStationHSUpcomingConfigurationOP11600 :
STRUCT
	{attribute 'OPC.UA.DA.Description' := 'Number of tools configured for the operation (0-200)'}
	ToolCapacityUsed			: UINT;
	
	{attribute 'OPC.UA.DA.Description' := 'IDs of upcoming tools'}
	{attribute 'OPC.UA.DA.StructuredType' := '1'}
	Tool 						: ARRAY [1..200] OF ToolX;

	{attribute 'OPC.UA.DA.Description' := 'Upcoming number of material configured for the operation (0-200)'}
	MaterialCapacityUsed		: UINT; 

	{attribute 'OPC.UA.DA.Description' := 'IDs OF upcoming material'}
	Material					: ARRAY [1..200] OF STRING(30);

END_STRUCT
END_TYPE

// ---- ECC/Cell_Unit_4/HeatAndSteam/OPC Data/Sub/Configuration/ST_OutputStationHSConfigurationOP11600.TcDUT
TYPE ST_OutputStationHSConfigurationOP11600 :
STRUCT
	{attribute 'OPC.UA.DA.Description' := 'Status variables for describing if the operation is restricted for specific SKUs'}
	{attribute 'OPC.UA.DA.StructuredType' := '1'}
	SKURestriction				: ST_SKURestriction;
	
	{attribute 'OPC.UA.DA.Description' := 'Possible tool amount for the operation'}
	ToolCapacity				: UINT;
	
	{attribute 'OPC.UA.DA.Description' := 'Possible material amount for the operation'}
	MaterialCapacity			: UINT;

	{attribute 'OPC.UA.DA.Description' := 'Current config for the operation'}
	{attribute 'OPC.UA.DA.StructuredType' := '1'}
	CurrentConfiguration		: ST_OutputStationHSCurrentConfigurationOP11600;

	{attribute 'OPC.UA.DA.Description' := 'Next config for the operation'}
	{attribute 'OPC.UA.DA.StructuredType' := '1'}
	UpcomingConfiguration		: ST_OutputStationHSUpcomingConfigurationOP11600;

	
END_STRUCT
END_TYPE

// ---- ECC/Cell_Unit_4/HeatAndSteam/OPC Data/Sub/Configuration/ST_OutputStationHSCurrentConfiguration.TcDUT
TYPE ST_OutputStationHSCurrentConfiguration :
STRUCT
// Handshake part
	{attribute 'OPC.UA.DA.Description' := 'Change acknowledge (0-255)'}
	ChangeAcknowledge		: UINT;
	
	{attribute 'OPC.UA.DA.Description' := 'Change status (0-255)'}
	ChangeStatus			: UINT;

// Data part
	{attribute 'OPC.UA.DA.Description' := 'Data changed (0-65536)'}
	DataChange				: UINT;
	
	{attribute 'OPC.UA.DA.Description' := 'Date and time'}
	DateTime				: DT;
	
	{attribute 'OPC.UA.DA.Description' := 'Configuration type (OPxxxxx or General)'}
	ConfigurationType		: STRING(7);
	
	{attribute 'OPC.UA.DA.Description' := 'General'}
	{attribute 'OPC.UA.DA.StructuredType' := '1'}
	General					: ST_OutputStationHSCurrentConfigurationGeneral;
	
	{attribute 'OPC.UA.DA.Description' := 'HeatAndSteam Step 1 Current Configuration'}
	{attribute 'OPC.UA.DA.StructuredType' := '1'}
	OP11600						: ST_InputStationHSConfigurationOP11600;
	
//	{attribute 'OPC.UA.DA.Description' := 'HeatAndSteam Step 2 Current Configuration'}
//	{attribute 'OPC.UA.DA.StructuredType' := '1'}
//	OP11601						: ST_InputStationHSConfigurationOP11601;	


END_STRUCT
END_TYPE

// ---- ECC/Cell_Unit_4/HeatAndSteam/OPC Data/Sub/Configuration/ST_OutputStationHSCurrentConfigurationGeneral.TcDUT
TYPE ST_OutputStationHSCurrentConfigurationGeneral :
STRUCT
	{attribute 'OPC.UA.DA.Description' := 'Dummy (for making struct visible on OPC UA'}
	Dummy						: BOOL;
END_STRUCT
END_TYPE

// ---- ECC/Cell_Unit_4/HeatAndSteam/OPC Data/Sub/Configuration/ST_OutputStationHSCurrentConfigurationOP11600.TcDUT
TYPE ST_OutputStationHSCurrentConfigurationOP11600 :
STRUCT
	{attribute 'OPC.UA.DA.Description' := 'Status variables for describing if the operation is restricted for specific SKUs'}
	{attribute 'OPC.UA.DA.StructuredType' := '1'}
	SKURestriction				: ST_SKURestriction;
	
	{attribute 'OPC.UA.DA.Description' := 'Possible tool amount for the operation'}
	ToolCapacity				: UINT;
	
	{attribute 'OPC.UA.DA.Description' := 'Number of tools configured for the operation (0-200)'}
	ToolCapacityUsed			: UINT;

	{attribute 'OPC.UA.DA.Description' := 'IDs of upcoming tools'}
	{attribute 'OPC.UA.DA.StructuredType' := '1'}
	Tool 						: ARRAY [1..200] OF ToolX;

	{attribute 'OPC.UA.DA.Description' := 'Status variables for current location and control mapping of tools'}
	{attribute 'OPC.UA.DA.StructuredType' := '1'}
	ToolMapping					: ARRAY [1..200] OF ToolXMapping;

	{attribute 'OPC.UA.DA.Description' := 'Possible material amount for the operation'}
	MaterialCapacity			: UINT;
	
	{attribute 'OPC.UA.DA.Description' := 'Upcoming number of material configured for the operation (0-200)'}
	MaterialCapacityUsed		: UINT; 

	{attribute 'OPC.UA.DA.Description' := 'IDs OF upcoming material'}
	Material					: ARRAY [1..200] OF STRING(30);

	{attribute 'OPC.UA.DA.Description' := 'Status variables for current location and control mapping of feeding material'}
	{attribute 'OPC.UA.DA.StructuredType' := '1'}
	MaterialMapping				: ARRAY [1..200] OF MaterialXMapping;
END_STRUCT
END_TYPE

// ---- ECC/Cell_Unit_4/HeatAndSteam/OPC Data/Sub/Configuration/ST_OutputStationHSUpcomingConfiguration.TcDUT
TYPE ST_OutputStationHSUpcomingConfiguration :
STRUCT
// Handshake part
	{attribute 'OPC.UA.DA.Description' := 'Change acknowledge (0-255)'}
	ChangeAcknowledge		: UINT;
	
	{attribute 'OPC.UA.DA.Description' := 'Change status (0-255)'}
	ChangeStatus			: UINT;

// Data part
	{attribute 'OPC.UA.DA.Description' := 'Data changed (0-65536)'}
	DataChange				: UINT;
	
	{attribute 'OPC.UA.DA.Description' := 'Date and time'}
	DateTime				: DT;
	
	{attribute 'OPC.UA.DA.Description' := 'Configuration type (OPxxxxx or General)'}
	ConfigurationType		: STRING(7);
	
	{attribute 'OPC.UA.DA.Description' := 'HeatAndSteam Step 1 Upcoming Configuration'}
	{attribute 'OPC.UA.DA.StructuredType' := '1'}
	OP11600						: ST_InputStationHSUpcomingConfigurationOP11600;
	
//	{attribute 'OPC.UA.DA.Description' := 'HeatAndSteam Step 2 Upcoming Configuration'}
//	{attribute 'OPC.UA.DA.StructuredType' := '1'}
//	OP11601						: ST_InputStationHSUpcomingConfigurationOP11601;	

END_STRUCT
END_TYPE

// ---- ECC/Cell_Unit_4/HeatAndSteam/OPC Data/Sub/Configuration/ST_OutputStationHSUpcomingConfigurationOP11600.TcDUT
TYPE ST_OutputStationHSUpcomingConfigurationOP11600 :
STRUCT
	{attribute 'OPC.UA.DA.Description' := 'Number of tools configured for the operation (0-200)'}
	ToolCapacityUsed			: UINT;

	{attribute 'OPC.UA.DA.Description' := 'IDs of upcoming tools'}
	{attribute 'OPC.UA.DA.StructuredType' := '1'}
	Tool 						: ARRAY [1..200] OF ToolX;

	{attribute 'OPC.UA.DA.Description' := 'Upcoming number of material configured for the operation (0-200)'}
	MaterialCapacityUsed		: UINT; 

	{attribute 'OPC.UA.DA.Description' := 'IDs OF upcoming material'}
	Material					: ARRAY [1..200] OF STRING(30);

END_STRUCT
END_TYPE

// ---- ECC/Cell_Unit_4/HeatAndSteam/OPC Data/Sub/Control/ST_InputStationHSControl.TcDUT
TYPE ST_InputStationHSControl :
STRUCT
	{attribute 'OPC.UA.DA.Description' := 'Station general configuration'}
	{attribute 'OPC.UA.DA.StructuredType' := '1'}
	General						: ST_InputStationHSControlGeneral;

	{attribute 'OPC.UA.DA.Description' := 'HeatAndSteam Control'}
	{attribute 'OPC.UA.DA.StructuredType' := '1'}
	OP11600						: ST_InputStationHSControlOP11600;

END_STRUCT
END_TYPE

// ---- ECC/Cell_Unit_4/HeatAndSteam/OPC Data/Sub/Control/ST_InputStationHSControlGeneral.TcDUT
TYPE ST_InputStationHSControlGeneral :
STRUCT
	{attribute 'OPC.UA.DA.Description' := 'TRUE to enable Simulation mode for HS device'}
	{attribute 'TcIgnorePersistent'}
	SimulationMode				: BOOL;
	
	{attribute 'OPC.UA.DA.Description' := 'Station idle time in minutes'}
	StationIdleTime				: UDINT;
	
END_STRUCT
END_TYPE

// ---- ECC/Cell_Unit_4/HeatAndSteam/OPC Data/Sub/Control/ST_InputStationHSControlOP11600.TcDUT
TYPE ST_InputStationHSControlOP11600 :
STRUCT
	{attribute 'OPC.UA.DA.Description' := 'OP11600 - Idle temperature C°'}
	IdleTemperature				: UINT;
	
	{attribute 'OPC.UA.DA.Description' := 'OP11600 - Idle Fan speed'}
	IdleFanSpeed				: UINT;
END_STRUCT
END_TYPE

// ---- ECC/Cell_Unit_4/HeatAndSteam/OPC Data/Sub/Information/ST_OutputHeaderCellInformationStationHS.TcDUT
TYPE ST_OutputHeaderCellInformationStationHS:// EXTENDS ST_OutputHeaderCellInformationStationX :
STRUCT
	{attribute 'OPC.UA.DA.Description' := 'Operation information'}
	{attribute 'OPC.UA.DA.StructuredType' := '1'}
	OperationInformation	: ARRAY [1..1] OF ST_OutputHeaderCellInformationStationInformationOperationInformationX;
	
	{attribute 'OPC.UA.DA.Description' := 'Station name'}
	StationName				: STRING;

	{attribute 'OPC.UA.DA.Description' := 'Station ID'}
	StationID				: STRING;
	
	{attribute 'OPC.UA.DA.Description' := 'PLC version'}
	NumberOfOperations		: UINT;
	
	{attribute 'OPC.UA.DA.Description' := 'Rework possible on this station'}
	Rework					: BOOL;

END_STRUCT
END_TYPE

// ---- ECC/Cell_Unit_4/HeatAndSteam/OPC Data/Sub/JobData/ST_InputStationHSJobData.TcDUT
TYPE ST_InputStationHSJobData :
STRUCT
	{attribute 'OPC.UA.DA.Description' := 'Change Request (0-255)'}
	{attribute 'TcIgnorePersistent'}
	ChangeRequest				: UINT;

	{attribute 'OPC.UA.DA.Description' := 'Job data type'}
	JobDataType				: STRING(7);

	{attribute 'OPC.UA.DA.Description' := '0: Undefined, 1: Different station, 2: Same station'}
	NextJobStation				: UINT;

			(* Might not be the same struct *)
	{attribute 'OPC.UA.DA.Description' := 'Job data HeatAndSteam Step 1'}
	{attribute 'OPC.UA.DA.StructuredType' := '1'}
	OP11600						: ST_InputStationHSJobDataOP11600;

//	{attribute 'OPC.UA.DA.Description' := 'Job data HeatAndSteam Step 2'}
//	{attribute 'OPC.UA.DA.StructuredType' := '1'}
//	OP11601						: ST_InputStationHSJobDataOP11601;
END_STRUCT
END_TYPE

// ---- ECC/Cell_Unit_4/HeatAndSteam/OPC Data/Sub/JobData/ST_InputStationHSJobDataOP11600.TcDUT
TYPE ST_InputStationHSJobDataOP11600 :
STRUCT
	{attribute 'OPC.UA.DA.Description' := 'Dynamic Tool'}
	{attribute 'OPC.UA.DA.StructuredType' := '1'}
	DynamicTool						: ARRAY [1..1] OF ToolX;

	{attribute 'OPC.UA.DA.Description' := 'Dynamic Material'}
	DynamicMaterial					: ARRAY [1..1] OF STRING(30);

	{attribute 'OPC.UA.DA.Description' := 'Temperature Target C°'}
	TemperatureTarget				: REAL;

	{attribute 'OPC.UA.DA.Description' := 'Temperature Max C°'}
	TemperatureMax					: REAL;
	
	{attribute 'OPC.UA.DA.Description' := 'Temperature Min C°'}
	TemperatureMin					: REAL;
	
	{attribute 'OPC.UA.DA.Description' := 'Time Max S'}
	TimeMax							: REAL;
	
	{attribute 'OPC.UA.DA.Description' := 'Time Min S'}
	TimeMin							: REAL;
	
	{attribute 'OPC.UA.DA.Description' := 'Steam Max'}
	SteamMax						: REAL;
	
	{attribute 'OPC.UA.DA.Description' := 'Steam Min'}
	SteamMin						: REAL;
	
	{attribute 'OPC.UA.DA.Description' := 'Air Max'}
	AirMax							: REAL;
	
	{attribute 'OPC.UA.DA.Description' := 'Air Min'}
	AirMin							: REAL;
	
	{attribute 'OPC.UA.DA.Description' := 'Profile'}
	Profile							: ARRAY [ 1..10] OF REAL;
	
END_STRUCT
END_TYPE

// ---- ECC/Cell_Unit_4/HeatAndSteam/OPC Data/Sub/JobData/ST_OutputStationHSJobData.TcDUT
TYPE ST_OutputStationHSJobData :
STRUCT
// HandShake part
	{attribute 'OPC.UA.DA.Description' := 'Change acknowledge (0-255)'}
	ChangeAcknowledge			: UINT;

	{attribute 'OPC.UA.DA.Description' := 'Data change status (0-255)'}
	ChangeStatus				: UINT;

// Data part
	{attribute 'OPC.UA.DA.Description' := 'Data changed (0-65536)'}
	DataChange					: UINT;
	
	{attribute 'OPC.UA.DA.Description' := 'Job data type'}
	JobDataType					: STRING(7);

	{attribute 'OPC.UA.DA.Description' := 'Job state (0: Undefined, 1: Idle, 2: Executing, 3: Completed'}
	JobState					: UINT;

	{attribute 'OPC.UA.DA.Description' := 'Job data HeatAndSteam Step 1'}
	{attribute 'OPC.UA.DA.StructuredType' := '1'}
	OP11600						: ST_InputStationHSJobDataOP11600;

//	{attribute 'OPC.UA.DA.Description' := 'Job data HeatAndSteam Step 2'}
//	{attribute 'OPC.UA.DA.StructuredType' := '1'}
//	OP11601						: ST_InputStationHSJobDataOP11601;
	
END_STRUCT
END_TYPE

// ---- ECC/Cell_Unit_4/HeatAndSteam/OPC Data/Sub/OperationalData/ST_OutputStationHSOperationalData.TcDUT
TYPE ST_OutputStationHSOperationalData :
STRUCT
// Handshake part
	{attribute 'OPC.UA.DA.Description' := 'Change acknowledged (0-255)'}
	ChangeAcknowledge	: UINT;

	{attribute 'OPC.UA.DA.Description' := 'Change status (0-255)'}
	ChangeStatus		: UINT;

// Data part	
	{attribute 'OPC.UA.DA.Description' := 'Data has changed (0-65536)'}
	DataChange			: UINT;
	
	{attribute 'OPC.UA.DA.Description' := 'General'}
	{attribute 'OPC.UA.DA.StructuredType' := '1'}
	General					: ST_OutputStationHSOperationalDataGeneral;
	
	{attribute 'OPC.UA.DA.Description' := 'OP11600'}
	{attribute 'OPC.UA.DA.StructuredType' := '1'}
	OP11600					: ST_OperationalDataOPxxxxx;
	
//	{attribute 'OPC.UA.DA.Description' := 'OP16101'}
//	{attribute 'OPC.UA.DA.StructuredType' := '1'}
//	OP11601					: ST_OperationalDataOPxxxxx;
END_STRUCT
END_TYPE

// ---- ECC/Cell_Unit_4/HeatAndSteam/OPC Data/Sub/OperationalData/ST_OutputStationHSOperationalDataGeneral.TcDUT
TYPE ST_OutputStationHSOperationalDataGeneral :
STRUCT
	{attribute 'OPC.UA.DA.Description' := 'Dummy (for making struct visible on OPC UA'}
	Dummy						: BOOL;
END_STRUCT
END_TYPE

// ---- ECC/Cell_Unit_4/HeatAndSteam/OPC Data/Sub/OperationalData/ST_OutputStationHSOperationalDataOP11600.TcDUT
TYPE ST_OutputStationHSOperationalDataOP11600 :
STRUCT
	{attribute 'OPC.UA.DA.Description' := 'Current number of tools where data is available'}
	NumberOfToolData			: UINT;

	{attribute 'OPC.UA.DA.Description' := 'Status variables for current operational data of tools'}
	{attribute 'OPC.UA.DA.StructuredType' := '1'}
	ToolData					: ARRAY [1..200] OF ToolDataX;

	{attribute 'OPC.UA.DA.Description' := 'Current number OF feeding material where data is available'}
	NumberOfMaterialData		: UINT;

	{attribute 'OPC.UA.DA.Description' := 'Status variables for current operational data of material'}
	{attribute 'OPC.UA.DA.StructuredType' := '1'}
	MaterialData				: ARRAY [1..200] OF MaterialDataX;

//	{attribute 'OPC.UA.DA.Description' := 'Status variables FOR current operational data of devices'}
//	{attribute 'OPC.UA.DA.StructuredType' := '1'}
//	DeviceData					: ST_Scanner_JobStatus;
	
END_STRUCT
END_TYPE

// ---- ECC/Cell_Unit_4/HeatAndSteam/OPC Data/Sub/Sustainability/ST_OutputStationHSSustainabilityData.TcDUT
TYPE ST_OutputStationHSSustainabilityData :
STRUCT
	{attribute 'OPC.UA.DA.Description' := 'Dummy (for making struct visible on OPC UA'}
	bDummy						: BOOL;
END_STRUCT
END_TYPE

// ---- ECC/Cell_Unit_4/OPC Data/Sub/ST_OutputCellOperationalDataGeneral.TcDUT
TYPE ST_OutputCellOperationalDataGeneral :
STRUCT
	{attribute 'OPC.UA.DA.Description' := 'E-Stop status'}
	bEStop						: BOOL;

	{attribute 'OPC.UA.DA.Description' := 'Doors status'}
	bDoors						: BOOL;

	{attribute 'OPC.UA.DA.Description' := 'Cell lights status'}
	bCellLight					: BOOL;

	{attribute 'OPC.UA.DA.Description' := 'PLC CPU Temperature'}
	rPLCCPUTemp					: REAL;

	{attribute 'OPC.UA.DA.Description' := 'Safety CPU Temperature'}
	rSafetyCPUTemp				: REAL;

	{attribute 'OPC.UA.DA.Description' := 'Station communication status'}
	bStationCommOK				: BOOL;

	{attribute 'OPC.UA.DA.Description' := 'Station PLC serial no'}
	sPLCSerial					: STRING;

	{attribute 'OPC.UA.DA.Description' := 'Station PLC mainboard serial no'}
	sPLCMBSerial				: STRING;

	{attribute 'OPC.UA.DA.Description' := 'CPU load/usage for the PLC runtime'}
	rPLCCPULoad					: REAL;

	{attribute 'OPC.UA.DA.Description' := 'CPU load/usage for the OS/system'}
	rOSCPULoad					: REAL;

	{attribute 'OPC.UA.DA.Description' := 'Actual CPU frequency'}
	rCPUFrequency				: REAL;

END_STRUCT
END_TYPE

// ---- ECC/Cell_Unit_4/ST_VehicleInHS.TcDUT
TYPE ST_VehicleInHS :
STRUCT
	sCarrierID		: STRING;	//ID of the carrier
	nVehicleNo		: UINT;		//Vehicle number
	fVelocity		: REAL; 	//Velocity setpoint station entered
	fCalculatedTIA	: REAL;		//Calculated time to arrival at staion 2 with current speed
	JobData			: ST_InputStationHSJobDataOP11600; //Job data for vehicle
END_STRUCT
END_TYPE

// ---- ECC/Components/E_ComponentErrors.TcDUT
{attribute 'qualified_only'}
{attribute 'strict'}
TYPE E_ComponentErrors :
(
	OK := 0,
	
	// Hardware
	HW_ECat_Not_OP,
	HW_UnderRange,
	HW_OverRange,
	HW_Limit1,
	HW_Limit2,
	HW_Error,
	HW_Internal_Error,
	HW_Watchdog,
	
	// Software
	SW_HiHi,
	SW_Hi,
	SW_LoLo,
	SW_Lo,
	SW_Internal_Error,
	
	// TwinsAFE
	TS_Stop,
	TS_Error,
	TS_FBError,
	TS_ComError,
	TS_ModuleError,
	TS_CMPError,
	TS_DeactivateError,
	TS_RestartError,
	TS_StopError,
	TS_Deactivated,
	TS_WaitCommError,
	
	Last
	
);
END_TYPE

// ---- ECC/Components/E_Cylinder_Cmd.TcDUT
{attribute 'strict'}
TYPE E_Cylinder_Cmd :
(
	Cyl_Cmd_None	:= 0,
	Cyl_Cmd_Fwd 	:= 1,
	Cyl_Cmd_Rev		:= 2
	
);
END_TYPE

// ---- ECC/Components/E_Cylinder_Sta.TcDUT
{attribute 'strict'}
TYPE E_Cylinder_Sta :
(
	Cyl_Sta_None	:= 0,
	Cyl_Sta_Fwd 	:= 1,
	Cyl_Sta_Rev		:= 2,
	Cyl_Sta_Err		:= 3
	
);
END_TYPE

// ---- ECC/Components/TwinSAFE/E_TwinSAFE_Group_Diag.TcDUT
/// TwinCAT Group Diag definitions
{attribute 'qualified_only'}
{attribute 'strict'}
TYPE E_TwinSAFE_Group_Diag :
(
	NO_ERROR		:= 0,
	FBERROR			:= 1,
	COMERROR		:= 2,
	MODULEERROR		:= 3,
	CMPERROR		:= 4,
	DEACTIVATEERROR	:= 5,
	RESTARTERROR	:= 6

) USINT;
END_TYPE

// ---- ECC/Components/TwinSAFE/E_TwinSAFE_Group_State.TcDUT
/// TwinCAT Group State definitions
{attribute 'qualified_only'}
{attribute 'strict'}
TYPE E_TwinSAFE_Group_State :
(
	RUN				:= 1,
	STOP			:= 2,
	ERROR			:= 4,
	RESET			:= 5,
	START			:= 6,
	STOPERROR		:= 7,
	DEACTIVE		:= 16,
	WAITCOMERROR	:= 17

) USINT;
END_TYPE

// ---- ECC/Components/TwinSAFE/E_TwinSAFE_Logic_State.TcDUT
/// TwinCAT Group Diag definitions
{attribute 'qualified_only'}
{attribute 'strict'}
TYPE E_TwinSAFE_Logic_State :
(
	OFFLINE			:= 0,	// gray
	RUN				:= 1,	// green
	STOP			:= 2,	// dark red
	SAFE			:= 3,	// red
	ERROR			:= 4,	// purple
	START			:= 6,	// blue
	PREPARE			:= 8,	// blue
	RESTORE			:= 10,	// blue
	PROJECT_CRC_OK	:= 11	// blue

) USINT;
END_TYPE

// ---- ECC/Tools/E_Method.TcDUT
{attribute 'qualified_only'}
{attribute 'strict'}
TYPE E_Method :
(
	Idle := 0,
	Busy,
	Error,
	Done
);
END_TYPE

// ---- ECC/Tools/E_OPCUA_Client_Seq.TcDUT
{attribute 'qualified_only'}
{attribute 'strict'}
TYPE E_OPCUA_Client_Seq :
(
	Idle := 0,
	CheckData,
	OpenSession,
	GetNameSpace,
	GetNode,
	Read,
	GetMethod,
	CallMethod,
	ReleaseNode,
	ReleaseMethod,
	CloseSession,
	Disconnect,
	Done

);
END_TYPE

// ---- ECC/Tools/LogToFile/ST_String_FIFO.TcDUT
TYPE ST_String_FIFO :
STRUCT
	Input_Pointer:INT;
	Output_Pointer:INT;
	Count:INT;
	Full:BOOL;
	DataTop:INT:=199; (*Change this to max array len *)
	DB: ARRAY[0..199] OF STRING(255);
END_STRUCT
END_TYPE

// ---- ECC/Tools/ST_OPC_Client_Data.TcDUT
TYPE ST_OPC_Client_Data :
STRUCT
	sRemoteVar		: STRING;
	eIdentifierType	: Tc3_PLCopen_OpcUa.E_UAIdentifierType;
	bWrite			: BOOL;	// TRUE to write
	iTargetSize		: UDINT;
	pTarget			: pVOID;
	bCommOK			: BOOL;
END_STRUCT
END_TYPE

// ---- ECC/Tools/ST_OutputArgInfoAndData_Basis.TcDUT
{attribute 'pack_mode' := '1'}
TYPE ST_OutputArgInfoAndData_Basis :
STRUCT
	nNumberOfOutputArguments: UDINT; // determined amount of output parameters
	nReserved: ARRAY[1..4] OF BYTE; // Reserved padding
	stOutputArgInfo: ARRAY[1..1] OF ST_UAMethodArgInfo; // number of output parameters - M_Mul has 1 output parameter 
END_STRUCT
END_TYPE

// ---- ECC/Tools/ST_Test.TcDUT
TYPE ST_Test :
STRUCT
	rTest	: REAL;
	iTest	: INT;
	bTest	: BOOL;
END_STRUCT
END_TYPE

// ---- ECC/TrackClient/Buffer Control/ST_BufferControl.TcDUT
TYPE ST_BufferControl :
STRUCT
	stData			: ST_MMBuffer;		// Data for vehicle
	iMoveCmdID		: UINT;				// Command ID for movement (to check status for movement)
END_STRUCT
END_TYPE

// ---- ECC/TrackClient/Enums/E_BufferState.TcDUT
{attribute 'qualified_only'}
{attribute 'strict'}
TYPE E_BufferState :
(
	Idle := 0,
	Waiting,
	CheckBuffer,
	MovePreBuffer,
	FinishedPre,
	MovePostBuffer,
	FinishedPost,
	MovePreToIn,
	FinishedPreToIn,
	MovePreToOut,
	FinishedPreToOut,
	MoveInToOut,
	FinishedInToOut,
	MoveOutToPost,
	FinishedOutToPost

);
END_TYPE

// ---- ECC/TrackClient/Enums/E_BufferStates.TcDUT
{attribute 'qualified_only'}
{attribute 'strict'}
TYPE E_BufferStates :
(
	Init := 0,
	Waiting,
	CheckBuffer,
	FindEmptyLocation,
	InsertIntoBuffer,
	CheckTicekts,
	SetTrafficLightRed,	
	SendOutOfBuffer,
	SetTrafficLightGreen
);
END_TYPE

// ---- ECC/TrackClient/Enums/E_PostBufferInState.TcDUT
{attribute 'qualified_only'}
{attribute 'strict'}
TYPE E_PostBufferInState :
(
	Waiting := 0,
	FindPosition,
	Infeed,
	ExtraVehicleRemove
);
END_TYPE

// ---- ECC/TrackClient/Enums/E_DecisionPointState.TcDUT
{attribute 'qualified_only'}
{attribute 'strict'}
TYPE E_DecisionPointState :
(
	Idle := 0,				// Wait state
	ReadVehicleData,		// Make sure vehicle data has been read from track server
	CheckTicket,			// Check if ticket is in the reservation buffer for this cell
	CheckPriority,			// Check if priority is correct
// If vehicle is to be used in this cell
	TakeOwnership,			// Take ownership of the vehicle (via. Track Server)
	WaitStationReady,		// Wait station ready
	MoveStation,			// Move vehicle to station (via. Track Server)
	WaitMoveStation,			// Wait for vehicle on station
	RemoveReservation,		// Remove ticket from reservation (via. Track Server)
// If it should not be used in this cell
	AddExtraToList,			// Add vehicle to extra list
	WaitStationEmpty,
	MoveNextCell,			// 
	WaitMoveNextCell		// 

);
END_TYPE

// ---- ECC/TrackClient/Enums/E_ExitPointState.TcDUT
{attribute 'qualified_only'}
{attribute 'strict'}
TYPE E_ExitPointState :
(
	Idle := 0,				// Wait state
	CheckBuffer,			// Check if there is vehicles ready for exit in post-buffer
	SetTrafficLightRd,		// 
	MoveVehicles,			// 
	SetTrafficLightGr		// 

);
END_TYPE

// ---- ECC/TrackClient/Enums/E_StationState.TcDUT
{attribute 'qualified_only'}
{attribute 'strict'}
TYPE E_StationState :
(
	Idle := 0,
	CheckStations,
	MoveToPostBuf,
	MoveToNextCell,
	ExtraVehicleRemove,	
	WaitMoveNextCell,
	AddReservation,			// Speciel handling for this cell - find and addReservation for this vehicle based on command data in buffer
	Done
);
END_TYPE

// ---- ECC/TrackClient/Enums/E_PostBufferOutState.TcDUT
{attribute 'qualified_only'}
{attribute 'strict'}
TYPE E_PostBufferOutState :
(
	Waiting := 0,
	CheckBuffer,
	FindVehicles,
	SetTrafficLightRed,	
	Outfeed,
	OutfeedStation,
	WaitOutfeedStation,
	SetTrafficLightGreen,
	CheckBufferSpace,
	Acumulate
);
END_TYPE

// ---- ECC/TrackClient/Station Control/E_StationBufferState.TcDUT
{attribute 'qualified_only'}
{attribute 'strict'}
TYPE E_StationBufferState :
(
	Idle := 0,
	CheckBuffer,
	StartMove,
	WaitMove
	
);
END_TYPE

// ---- ECC/TrackClient/Station Control/E_StationInOutState.TcDUT
{attribute 'qualified_only'}
{attribute 'strict'}
TYPE E_StationInOutState :
(
	Idle := 0,
	Check,
	StartMoveOut,
	WaitMoveOut,
	StartMoveIn,
	WaitMoveIn
	
);
END_TYPE

// ---- ECC/TrackClient/Station Control/ST_StationControlData.TcDUT
TYPE ST_StationControlData :
STRUCT
	nTicket			: UINT;
	nTicketSize		: UINT;
	nCarrierID		: UINT;
	nPriority		: UINT;
END_STRUCT
END_TYPE

// ---- ReadConfigFile/DUT_STRUCT_VARIABLES.TcDUT
TYPE DUT_STRUCT_VARIABLES :
STRUCT
	sEnvironment		:STRING;
	sCellName			:STRING;
	sIpAddress			:STRING;
	sAmsNetId			:STRING;
	sOpcUaURL			:STRING;
//	sUhfRfidOpcUaURL	:STRING;
//	sHfRfidOpcUaURL		:STRING;
	sStation1			:STRING;
	sTrackserver		:STRING;
	sTrackserver_AMS	:STRING;
//	sStation2			:STRING;
//	sStation3			:STRING;
//	sStation4			:STRING;
//	sRelease			:STRING;
//	sCommitID			:STRING;
//	sTag				:STRING;
END_STRUCT
END_TYPE

// ---- ECC/Basic/GVL_BASIC.TcGVL
VAR_GLOBAL
	Units		: FB_Units;
	g_rPLCScan_S		: REAL;				// [s] PLC scantime
	g_iPLCScan_MS		: UINT;				// [ms] PLC scantime
END_VAR

// ---- ECC/Basic/TrackClient/GVLs/GlobalConstants.TcGVL
VAR_GLOBAL CONSTANT
	(* Bridge related *)
	MM_MAX_NUMBER_OF_PATH_ELEMENTS			: UINT		:= 30;			(* The maximum number of paths that the server should handle. OBS!: If mulitible cells owns a path, they will each be defined as a path element. *)						
	MM_MAX_NUMBER_OF_STATION_ELEMENTS		: UINT		:= 20;			(* The maximum number of stations that the server should handle. OBS!: If mulitible stations are linked to a MM Station, they will each be defined as a station element. *)		
	MM_MAX_NUMBER_OF_TRAFFICLIGHT_ELEMENTS	: UINT		:= 20;			(* The maximum number of trafficlights that the server should handle. OBS!: If mulitible traffic lights are linked to a MM traffic light, they will each be defined as a traffic light element. *)
																		(* Maximum in the MagneMotion system is 32 Traffic Lights! *)		
	MM_MAX_BUFFER_INDEX						: USINT		:= 20;			(* The maximum number of pre-buffer or post-buffer indexes each station is allowed to have. *)		
	MM_MAX_NUMBER_OF_VEHICLE_ELEMENTS		: UINT		:= 50;			(* The maximum number of vehicles that the track server should handle. *)
	MM_MAX_NUMBER_OF_VEHICLE_CONFIGURATIONS	: UINT		:= 50;			(* The maximum number of vehicles configurations that the track server should handle. *)
	MM_MAX_NUMBER_OF_CELL_ELEMENTS			: UINT		:= 20;			(* The maxmimum nubmer of cells in the system *)			
	MM_MAX_RESERVATIONLIST_ELEMENTS			: UINT		:= 20;			(* The maximum number of reservations in the cell reservation list *)			
	MM_BUFFER_DISTANCE						: REAL		:= 50.0;		(* Distance between buffer points in pre/post buffers *)

END_VAR

// ---- ECC/Components/GVL_Components.TcGVL
VAR_GLOBAL
	bTestMode			: BOOL;	// TEST mode activated
	{attribute 'OPC.UA.DA':='1'}
	{attribute 'OPC.UA.DA.Access' := '3'}
	{attribute 'OPC.UA.DA.Description' := 'Use Simulation mode'}
	bSIMUMode			: BOOL;	// TRUE to activate Simulation mode
END_VAR

// ---- ECC/Tools/LogToFile/GVL_Log.TcGVL
VAR_GLOBAL
	LogToTextBuffer		: ST_String_FIFO;	// Text log
	fbLocalTime			: FB_LocalSystemTime;
END_VAR

// ---- GVLs/GVL.TcGVL
VAR_GLOBAL CONSTANT
	{attribute 'OPC.UA.DA':='1'}
	{attribute 'OPC.UA.DA.Access' := '1'}
	{attribute 'OPC.UA.DA.Description' := 'SW Version'}
	sSWVersion			: STRING := '0.1';

	iNoOfRecipeData		: UINT := 100;
END_VAR
VAR_GLOBAL
	bLogToOutputWindow	: BOOL;		// if TRUE it will log all logs to file AND to output window
	
	// read config file
	sString				:ARRAY[0..15] OF STRING(255);
	sVars				:DUT_STRUCT_VARIABLES;
END_VAR

// ---- POUs/MAIN.TcPOU
PROGRAM MAIN
VAR
	// OPC UA mapper for cell
	{attribute 'OPC.UA.DA':='1'}
	Bridge					: FB_OPC_Cell_Unit_4;

// Cell handling, PackML etc.
	fbUnit4					: FB_Cell_Unit_4;

// Log to file
	fbLogToFile				: FB_LogToFile;
	
//	LicenseState	AT %I*	: UINT;
	bInitDone 				: BOOL;
	
	// read config file
	fbReadFile				:FB_ReadFile;
	
END_VAR

// read config file
fbReadFile();

M_Init();

// Cell handling
fbUnit4(stModeStateIn := Bridge.Input.Cell.ModeState, 
		stModeStateOut := Bridge.Output.Cell.ModeState,
		stOEE := Bridge.Output.Cell.OEE,
		stErrorWarning := Bridge.Output.Cell.ErrorWarning,
		bResetEStop:= Bridge.P_bResetEStop,
		bLockDoor:= Bridge.P_bLockDoors, 
		bUnlockDoor:= Bridge.P_bUnlockDoors, 
		bCellLight:= Bridge.P_bCellLight,
		iHeartBeatFromMES:= Bridge.P_iHeartBeat,
		Input := Bridge.Input,		// Bridge Data Inputs
		Output := Bridge.Output, 	// Bridge Data Outputs
		bModeChangeInProcess=> 	);
		

// OPC handling
	// OPC handling
	Bridge.P_bEStop := fbUnit4.bEStopOK; 
	Bridge.P_bDoors := fbUnit4.bDoorsOK;
	Bridge.P_bCellLight := fbUnit4.bCellLightOn;
	Bridge.P_rPLCCPUTemp := fbUnit4.rCPUTemp;
	Bridge.P_rSafetyCPUTemp := fbUnit4.rSafetyTemp;
	Bridge.P_sPLCSerial := fbUnit4.sSerialIPC;
	Bridge.P_sPLCMBSerial := fbUnit4.sSerialMB;
	Bridge.P_bStationCommOK := NOT fbUnit4.bStationCommError;
	Bridge.P_iHeartBeat := fbUnit4.iHeartBeatToMES;
	Bridge.P_rOSCPULoad := fbUnit4.rCPULoad;
	Bridge.P_rPLCCPULoad := fbUnit4.rCPULoadPLC;
	Bridge.P_rCPUFrequency := fbUnit4.rCPUFrequency;
	Bridge();

//File logging
fbLocalTime(
	sNetID:= '', 
	bEnable:= TRUE, 
	dwCycle:= 5, 
	dwOpt:= 0, 
	tTimeout:=DEFAULT_ADS_TIMEOUT );	
	
fbLogToFile(Busy=> );

METHOD M_Init : BOOL
VAR_INPUT
END_VAR
// Init
IF (NOT bInitDone) THEN

	bInitDone := TRUE;
END_IF
END_METHOD

END_PROGRAM

// ---- ECC/Cell_Unit_4/FB_OPC_Cell_Unit_4.TcPOU
FUNCTION_BLOCK FB_OPC_Cell_Unit_4 //EXTENDS FB_OPC_Basic IMPLEMENTS ITF_OPC_Basic
VAR_OUTPUT
	{attribute 'OPC.UA.DA':='1'}
	{attribute 'OPC.UA.DA.Access' := '1'}
	{attribute 'OPC.UA.DA.Description' := 'Cell 4 bridge output data'}
	{attribute 'OPC.UA.DA.DisplayName' := 'Cell 4 bridge output data'}
	{attribute 'OPC.UA.DA.StructuredType' := '1'}
	Output			: ST_Output;

END_VAR
VAR_OUTPUT PERSISTENT
	{attribute 'OPC.UA.DA':='1'}
	{attribute 'OPC.UA.DA.Access' := '3'}
	{attribute 'OPC.UA.DA.Description' := 'Cell 4 bridge input data'}
	{attribute 'OPC.UA.DA.DisplayName' := 'Cell 4 bridge input data'}
	{attribute 'OPC.UA.DA.StructuredType' := '1'}
	Input			: ST_Input;

END_VAR
VAR
	bInitDone					: BOOL;
	bInhibitOPCUpdate			: BOOL;		// Set to TRUE to stop updating values from OPC structures
END_VAR

// Init values
M_Init();

// Data change status handling for cell
IF (NOT Input.Cell.AdditionalData.Settings.DataChangeStatusModeStateEnable) THEN
	Input.Cell.AdditionalData.MESHandShakes.DataChangeStatusModeState := Output.Cell.ModeState.DataChange;
END_IF
IF (NOT Input.Cell.AdditionalData.Settings.DataChangeStatusOEEEnable) THEN
	Input.Cell.AdditionalData.MESHandShakes.DataChangeStatusOEE := Output.Cell.OEE.DataChange;
END_IF
IF (NOT Input.Cell.AdditionalData.Settings.DataChangeStatusErrorWarningEnable) THEN
	Input.Cell.AdditionalData.MESHandShakes.DataChangeStatusErrorWarning := Output.Cell.ErrorWarning.DataChange;
END_IF
IF (NOT Input.Cell.AdditionalData.Settings.DataChangeStatusOperationalDataEnable) THEN
	Input.Cell.AdditionalData.MESHandShakes.DataChangeStatusOperationalData := Output.Cell.OperationalData.DataChange;
END_IF
	
// Data change status handling for Station 1
IF (NOT Input.Station.Station1.AdditionalData.Settings.DataChangeStatusModeStateEnable) THEN
	Input.Station.Station1.AdditionalData.MESHandShakes.DataChangeStatusModeState := Output.Station.Station1.ModeState.DataChange;
END_IF
IF (NOT Input.Station.Station1.AdditionalData.Settings.DataChangeStatusJobDataEnable) THEN
	Input.Station.Station1.AdditionalData.MESHandShakes.DataChangeStatusJobData := Output.Station.Station1.JobData.DataChange;
END_IF
IF (NOT Input.Station.Station1.AdditionalData.Settings.DataChangeStatusOEEEnable) THEN
	Input.Station.Station1.AdditionalData.MESHandShakes.DataChangeStatusOEE := Output.Station.Station1.OEE.DataChange;
END_IF
IF (NOT Input.Station.Station1.AdditionalData.Settings.DataChangeStatusErrorWarningEnable) THEN
	Input.Station.Station1.AdditionalData.MESHandShakes.DataChangeStatusErrorWarning := Output.Station.Station1.ErrorWarning.DataChange;
END_IF
IF (NOT Input.Station.Station1.AdditionalData.Settings.DataChangeStatusCurrentConfigurationEnable) THEN
	Input.Station.Station1.AdditionalData.MESHandShakes.DataChangeStatusCurrentConfiguration := Output.Station.Station1.CurrentConfiguration.DataChange;
END_IF
IF (NOT Input.Station.Station1.AdditionalData.Settings.DataChangeStatusUpcomingConfigurationEnable) THEN
	Input.Station.Station1.AdditionalData.MESHandShakes.DataChangeStatusUpcomingConfiguration := Output.Station.Station1.UpcomingConfiguration.DataChange;
END_IF
IF (NOT Input.Station.Station1.AdditionalData.Settings.DataChangeStatusOperationalDataEnable) THEN
	Input.Station.Station1.AdditionalData.MESHandShakes.DataChangeStatusOperationalData := Output.Station.Station1.OperationalData.DataChange;
END_IF

// Data change status handling for Station 1
IF (NOT Input.Transport.AdditionalData.Settings.DataChangeStatusTransportStatusEnable) THEN
	Input.Transport.AdditionalData.MESHandShakes.DataChangeStatusTransportStatus := Output.Transport.Status.DataChange;
END_IF
IF (NOT Input.Transport.AdditionalData.Settings.DataChangeStatusTransportMappingEnable) THEN
	Input.Transport.AdditionalData.MESHandShakes.DataChangeStatusTransportMapping := Output.Transport.Mapping.DataChange;
END_IF

METHOD M_init : BOOL
VAR_INPUT
END_VAR
IF (NOT bInitDone) THEN
	bInitDone := TRUE;
END_IF
END_METHOD

PROPERTY PUBLIC P_bCellLight : BOOL
GET
P_bCellLight := Input.Cell.Control.EnableCellLight;
END_GET
SET
Output.Cell.OperationalData.General.bCellLight := P_bCellLight;
END_SET
END_PROPERTY

PROPERTY PUBLIC P_bDoors : BOOL
SET
Output.Cell.OperationalData.General.bDoors := P_bDoors;
END_SET
END_PROPERTY

PROPERTY PUBLIC P_bEStop : BOOL
GET
P_bEStop := Output.Cell.OperationalData.General.bEStop;
END_GET
SET
Output.Cell.OperationalData.General.bEStop := P_bEStop;
END_SET
END_PROPERTY

PROPERTY P_bLockDoors : BOOL
GET
P_bLockDoors := Input.Cell.Control.LockDoors;
END_GET
END_PROPERTY

PROPERTY P_bResetEStop : BOOL
GET
P_bResetEStop := Input.Cell.Control.ResetEStop;
END_GET
END_PROPERTY

PROPERTY PUBLIC P_bStationCommOK : BOOL
GET
P_bStationCommOK := Output.Cell.OperationalData.General.bStationCommOK;
END_GET
SET
Output.Cell.OperationalData.General.bStationCommOK := P_bStationCommOK;
END_SET
END_PROPERTY

PROPERTY P_bUnlockDoors : BOOL
GET
P_bUnlockDoors := Input.Cell.Control.UnlockDoors;
END_GET
END_PROPERTY

PROPERTY PUBLIC P_iHeartBeat : UINT
GET
P_iHeartBeat := Input.Header.HeartBeat;
END_GET
SET
Output.Header.HeartBeat := P_iHeartBeat;
END_SET
END_PROPERTY

PROPERTY PUBLIC P_rCPUFrequency : REAL
GET
P_rCPUFrequency := Output.Cell.OperationalData.General.rCPUFrequency;
END_GET
SET
Output.Cell.OperationalData.General.rCPUFrequency := P_rCPUFrequency;
END_SET
END_PROPERTY

PROPERTY PUBLIC P_rOSCPULoad : REAL
GET
P_rOSCPULoad := Output.Cell.OperationalData.General.rOSCPULoad;
END_GET
SET
Output.Cell.OperationalData.General.rOSCPULoad := P_rOSCPULoad;
END_SET
END_PROPERTY

PROPERTY PUBLIC P_rPLCCPULoad : REAL
GET
P_rPLCCPULoad := Output.Cell.OperationalData.General.rPLCCPULoad;
END_GET
SET
Output.Cell.OperationalData.General.rPLCCPULoad := P_rPLCCPULoad;
END_SET
END_PROPERTY

PROPERTY PUBLIC P_rPLCCPUTemp : REAL
GET
P_rPLCCPUTemp := Output.Cell.OperationalData.General.rPLCCPUTemp;
END_GET
SET
Output.Cell.OperationalData.General.rPLCCPUTemp := P_rPLCCPUTemp;
END_SET
END_PROPERTY

PROPERTY PUBLIC P_rSafetyCPUTemp : REAL
GET
P_rSafetyCPUTemp := Output.Cell.OperationalData.General.rSafetyCPUTemp;
END_GET
SET
Output.Cell.OperationalData.General.rSafetyCPUTemp := P_rSafetyCPUTemp;
END_SET
END_PROPERTY

PROPERTY PUBLIC P_sPLCMBSerial : STRING
GET

P_sPLCMBSerial := Output.Cell.OperationalData.General.sPLCMBSerial;
END_GET
SET
Output.Cell.OperationalData.General.sPLCMBSerial := P_sPLCMBSerial;
END_SET
END_PROPERTY

PROPERTY PUBLIC P_sPLCSerial : STRING
GET
P_sPLCSerial := Output.Cell.OperationalData.General.sPLCSerial;
END_GET
SET
Output.Cell.OperationalData.General.sPLCSerial := P_sPLCSerial;
END_SET
END_PROPERTY

END_FUNCTION_BLOCK

// ---- ECC/Cell_Unit_4/FB_Cell_Unit_4.TcPOU
FUNCTION_BLOCK FB_Cell_Unit_4 EXTENDS FB_Cell_Basic
VAR_INPUT
END_VAR
VAR_OUTPUT
	bError						: BOOL;
	iErrorID					: BOOL;
END_VAR
VAR_IN_OUT
	// Bridge data
	Input						: ST_Input;
	Output						: ST_Output;
END_VAR
VAR
// Local vars
	eSeq						: E_VehicleOnStation;
	tonSeqTimer					: TON;
	aVehiclesStationFIFO		: ARRAY[1..10] OF ST_VehicleInHS;
	aDummyVehicleStationData	: ST_VehicleInHS;
	fDistanceStation2Station	: REAL; //Distance between stations

	stDeviceInfo				: ST_DeviceIdentification;			// Device information such as serial no.
	stVehicleDataOnStation		: ST_ReadVehicleData;
	nPLCVersion					: UINT:=0;
	nScannerInterfaceVersion	: UINT:=0;	
	bInitDone					: BOOL;
	bVehicleEnterStationOS	 	: BOOL;
	bVehicleMoveToStation		: BOOL;
	iRes						: INT;
	diFifoLogTimer				: UINT;
	diVehiclesInDevice			: UINT;
	
	tonVehicleDataRead			: TON;	// To trig reading of data for vehicles in the FIFO buffer

// FunctionBlocks:
	fbStationINHeatAndSteam		: FB_HeatAndSteamIN;
	fbStationOUTHeatAndSteam	: FB_HeatAndSteamOUT;
	fbTrack						: FB_TrackClient;
	
// Start op procedure
	bBypassTrack	:	BOOL;
	nCheckValid		:	UINT;
	nIndx			:	UINT;
	nIndxStart		:	UINT;
	nIndxDone		:	UINT;
	fVel			:	REAL;
	fAcc			:	REAL;
	bStartupPrd		:	BOOL;
	
// Error / Warnings
	iST1ErrWarDataChange	: UINT;
	iST2ErrWarDataChange	: UINT;
	iTCErrWarDataChange		: UINT;
END_VAR

SUPER^(	stModeStateIn := Input.Cell.ModeState,
		stModeStateOut := Output.Cell.ModeState,
		stOEE := Output.Cell.OEE,
		stErrorWarning := Output.Cell.ErrorWarning);

// Init FB's
M_Init();

// Run components
M_Components();
		
// Device controller
M_Device_Sequence();

// Error and warnings
M_ErrorWarning();

//Sustainability Data
M_SustainabilityDataHandling();

//Clear all ticket data
IF Input.Cell.AdditionalData.ClearAll THEN
	Input.Cell.AdditionalData.ClearAll R= M_ClearAll();
END_IF

// Update PackML state/modes variables from local values
bEStopOK := TRUE;
bStartLocal;
bStopLocal;
bClearLocal;
bResetLocal := ((eCurrentState = E_PMLState.ePMLState_Complete) AND (eCommand = E_PMLCommand.ePMLCommand_Undefined)); // Automatic back to Idle when finished
bHoldLocal;
bProductionLocal;
bManualLocal;

{attribute 'object_name' := 'M_Aborted'}
METHOD M_Aborted
END_METHOD

{attribute 'object_name' := 'M_Aborting'}
METHOD M_Aborting
// Stop all moving parts


// Abort is handled internally in Brushing Station FB, follows Cell unit state!
//IF (fbScanner1.stModeStateOut.CurrentMode = E_PML_State.Aborted) THEN
//	M_StateComplete();	
//END_IF


// No moving parts, go straight to nest state
//eCommand := E_PML_Command.Undefined;
M_StateComplete();
END_METHOD

METHOD PROTECTED M_CarrierFinishInfeedToTrack : BOOL
VAR_INPUT
END_VAR

// TODO!!!
M_CarrierFinishInfeedToTrack := TRUE;
END_METHOD

METHOD PROTECTED M_CarrierFinishOutfeedToTrack : BOOL
VAR_INPUT
END_VAR

// TODO!!!
M_CarrierFinishOutfeedToTrack := TRUE;
END_METHOD

METHOD PROTECTED M_CarrierReadyInfeedFromTrack : BOOL
VAR_INPUT
END_VAR

// TODO!!!
M_CarrierReadyInfeedFromTrack := FALSE;
END_METHOD

METHOD PROTECTED M_CarrierReadyOutfeedFromTrack : BOOL
VAR_INPUT
END_VAR

// TODO!!!
M_CarrierReadyOutfeedFromTrack := TRUE;
END_METHOD

METHOD M_ClearAll : BOOL
VAR_INPUT
END_VAR
VAR
	i : USINT;
END_VAR
//Clear all ticket data on cell from OPC command

//Clear Station(s) and TrackClient
IF fbStationINHeatAndSteam.M_ClearAll() AND fbStationOUTHeatAndSteam.M_ClearAll() THEN
	M_ClearAll := fbTrack.M_ClearAll();
END_IF
	
//Clear Cell
IF M_ClearAll THEN
	 eSeq := E_VehicleOnStation.Idle;
	 
	 //Clean out FIFO
	FOR i := 1 TO 9 DO
		aVehiclesStationFIFO[i] := aDummyVehicleStationData;
	END_FOR	
	F_Logfile('Cell - All data cleared!');
END_IF
END_METHOD

{attribute 'object_name' := 'M_Clearing'}
METHOD M_Clearing
// Reset safety system

//fbScanner1.nCellStateCmd := E_PML_Command.Clear;

//fbTrack.bReset := TRUE;

//IF ((fbScanner1.stModeStateOut.CurrentMode = E_PML_State.idle) OR (fbScanner1.stModeStateOut.CurrentMode = E_PML_State.stopped)) THEN
//	M_StateComplete();
	
//	fbTrack.bReset := FALSE;
//END_IF
//eCommand := E_PML_Command.Undefined;
M_StateComplete();
END_METHOD

{attribute 'object_name' := 'M_Complete'}
METHOD M_Complete
END_METHOD

{attribute 'object_name' := 'M_Completing'}
METHOD M_Completing

VAR
	sLowHighUpperID : STRING;	
	iRes			: INT;
END_VAR

//eCommand := E_PML_Command.Undefined;
M_StateComplete();
END_METHOD

METHOD PROTECTED M_Components : BOOL
VAR_INPUT
END_VAR
VAR
END_VAR
// Run component blocks
END_METHOD

METHOD M_Device_Sequence
VAR_INPUT
END_VAR
VAR
	i			: UINT;
	iRes		: INT;
	bMoveToNext	: BOOL;
END_VAR
// Heart beat
iHeartBeatFromMES := Input.Header.HeartBeat;
Output.Header.HeartBeat := iHeartBeatToMES;

